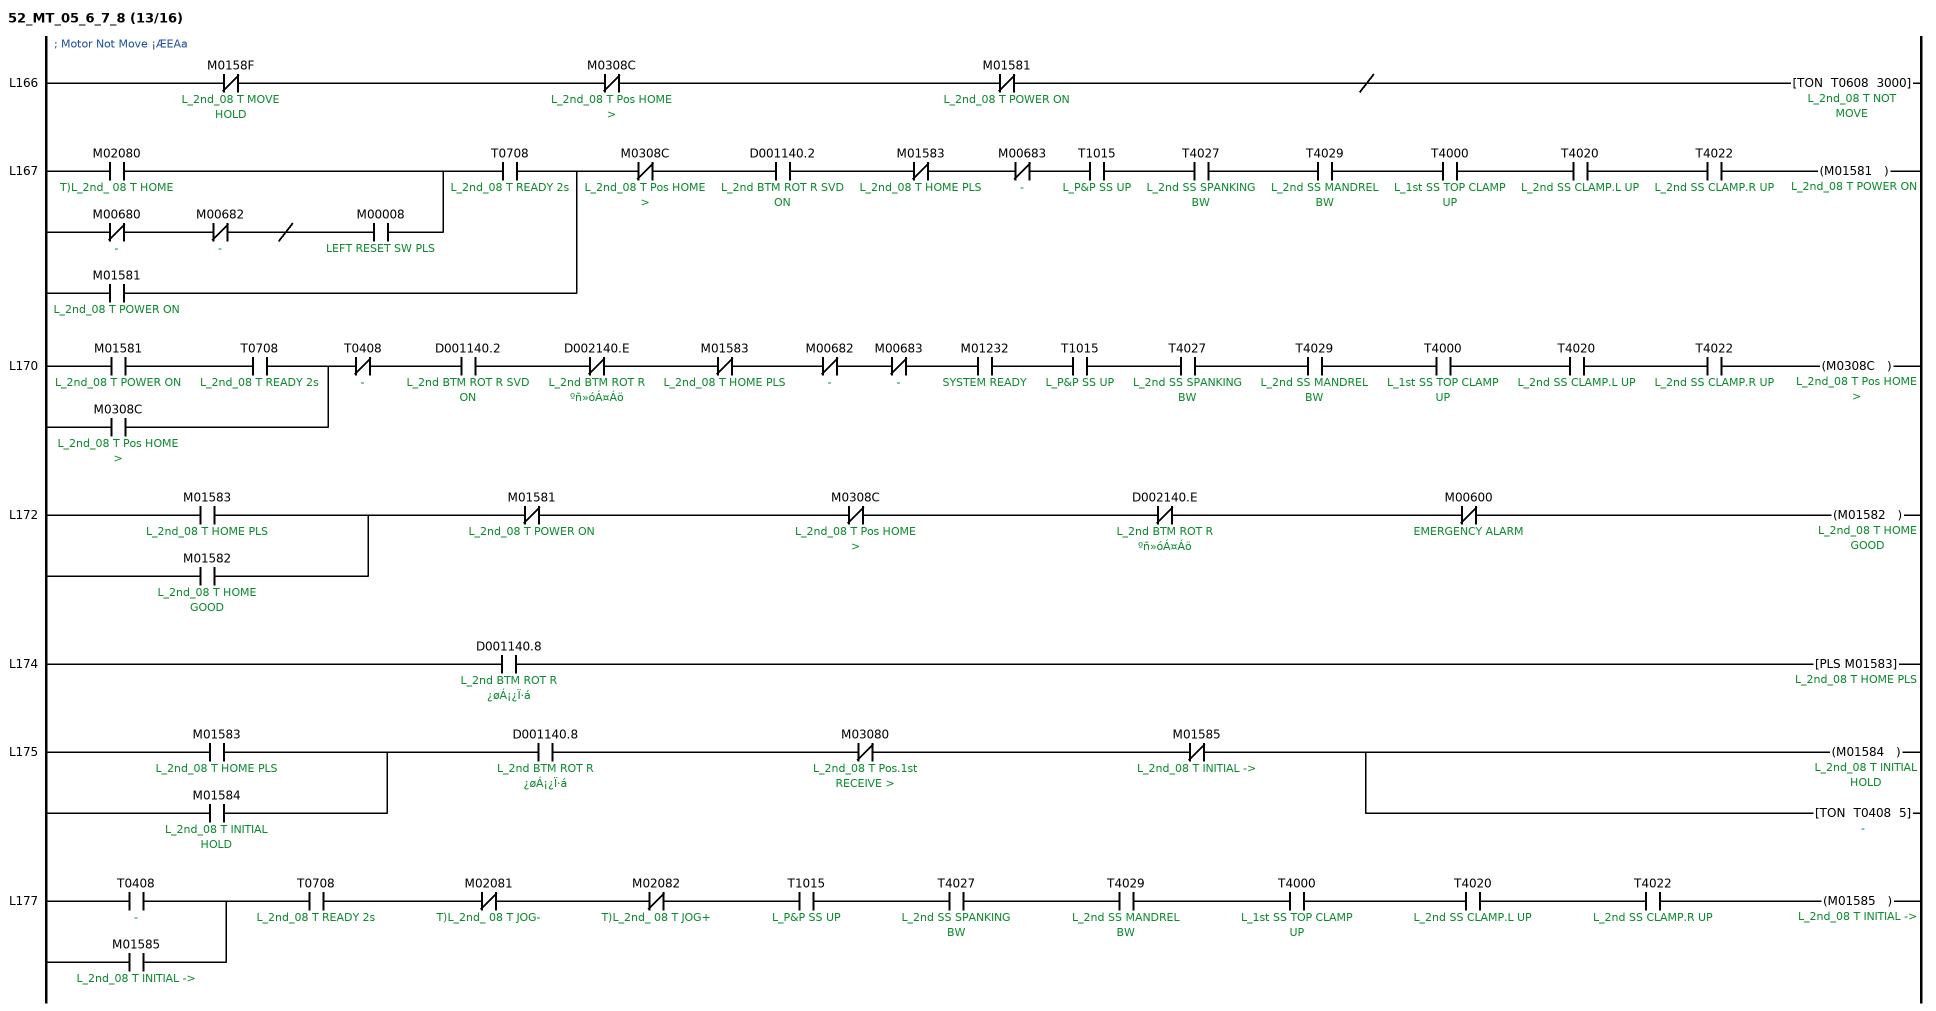
[picture p288: 52_MT_05_6_7_8 rungs L166-L177]
; L166
LOAD NOT  M0158F	// L_2nd_08 T MOVE HOLD
AND NOT   M0308C	// L_2nd_08 T Pos HOME >
AND NOT   M01581	// L_2nd_08 T POWER ON
NOT
TON       T0608 3000	// L_2nd_08 T NOT MOVE
// output comment: Motor Not Move ¡ÆEAa
; L167
LOAD      M02080	// T)L_2nd_ 08 T HOME
LOAD NOT  M00680	// -
AND NOT   M00682	// -
NOT
AND       M00008	// LEFT RESET SW PLS
OR LOAD
AND       T0708	// L_2nd_08 T READY 2s
OR        M01581	// L_2nd_08 T POWER ON
AND NOT   M0308C	// L_2nd_08 T Pos HOME >
AND       D001140.2	// L_2nd BTM ROT R SVD ON
AND NOT   M01583	// L_2nd_08 T HOME PLS
AND NOT   M00683	// -
AND       T1015	// L_P&P SS UP
AND       T4027	// L_2nd SS SPANKING BW
AND       T4029	// L_2nd SS MANDREL BW
AND       T4000	// L_1st SS TOP CLAMP    UP
AND       T4020	// L_2nd SS CLAMP.L UP
AND       T4022	// L_2nd SS CLAMP.R UP
OUT       M01581	// L_2nd_08 T POWER ON
; L170
LOAD      M01581	// L_2nd_08 T POWER ON
AND       T0708	// L_2nd_08 T READY 2s
OR        M0308C	// L_2nd_08 T Pos HOME >
AND NOT   T0408	// -
AND       D001140.2	// L_2nd BTM ROT R SVD ON
AND NOT   D002140.E	// L_2nd BTM ROT R ºñ»óÁ¤Áö
AND NOT   M01583	// L_2nd_08 T HOME PLS
AND NOT   M00682	// -
AND NOT   M00683	// -
AND       M01232	// SYSTEM READY
AND       T1015	// L_P&P SS UP
AND       T4027	// L_2nd SS SPANKING BW
AND       T4029	// L_2nd SS MANDREL BW
AND       T4000	// L_1st SS TOP CLAMP    UP
AND       T4020	// L_2nd SS CLAMP.L UP
AND       T4022	// L_2nd SS CLAMP.R UP
OUT       M0308C	// L_2nd_08 T Pos HOME >
; L172
LOAD      M01583	// L_2nd_08 T HOME PLS
OR        M01582	// L_2nd_08 T HOME GOOD
AND NOT   M01581	// L_2nd_08 T POWER ON
AND NOT   M0308C	// L_2nd_08 T Pos HOME >
AND NOT   D002140.E	// L_2nd BTM ROT R ºñ»óÁ¤Áö
AND NOT   M00600	// EMERGENCY ALARM
OUT       M01582	// L_2nd_08 T HOME GOOD
; L174
LOAD      D001140.8	// L_2nd BTM ROT R ¿øÁ¡¿Ï·á
OUTP      M01583	// L_2nd_08 T HOME PLS
; L175
LOAD      M01583	// L_2nd_08 T HOME PLS
OR        M01584	// L_2nd_08 T INITIAL HOLD
AND       D001140.8	// L_2nd BTM ROT R ¿øÁ¡¿Ï·á
AND NOT   M03080	// L_2nd_08 T Pos.1st RECEIVE >
AND NOT   M01585	// L_2nd_08 T INITIAL ->
OUT       M01584	// L_2nd_08 T INITIAL HOLD
TON       T0408 5	// -
; L177
LOAD      T0408	// -
OR        M01585	// L_2nd_08 T INITIAL ->
AND       T0708	// L_2nd_08 T READY 2s
AND NOT   M02081	// T)L_2nd_ 08 T JOG-
AND NOT   M02082	// T)L_2nd_ 08 T JOG+
AND       T1015	// L_P&P SS UP
AND       T4027	// L_2nd SS SPANKING BW
AND       T4029	// L_2nd SS MANDREL BW
AND       T4000	// L_1st SS TOP CLAMP    UP
AND       T4020	// L_2nd SS CLAMP.L UP
AND       T4022	// L_2nd SS CLAMP.R UP
OUT       M01585	// L_2nd_08 T INITIAL ->

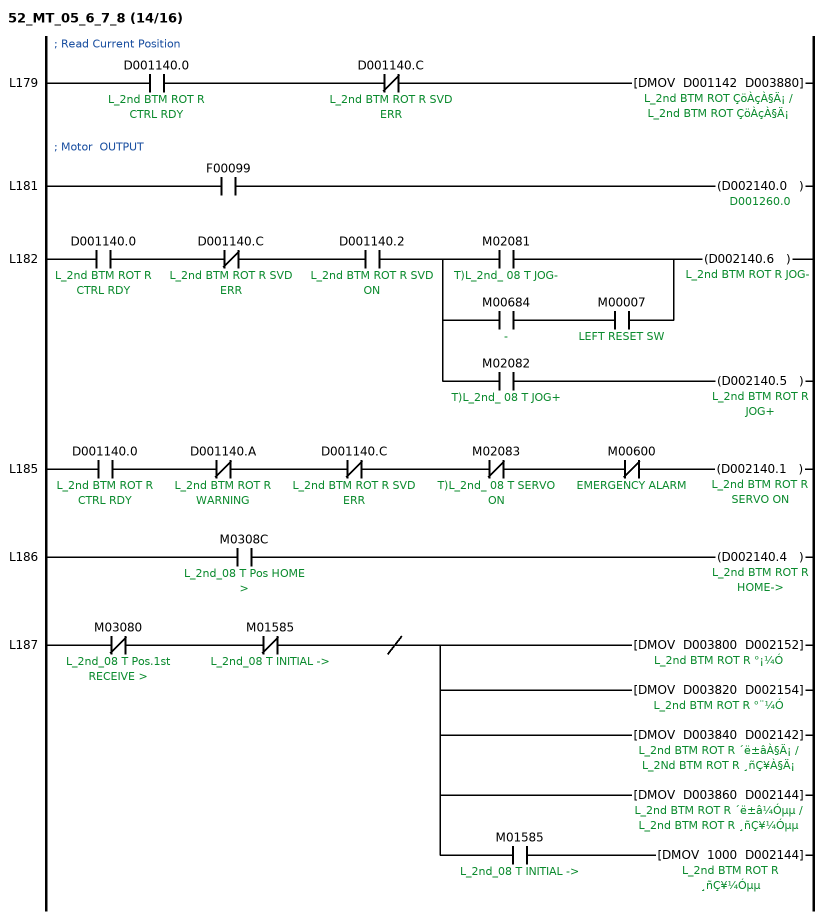
; L179
LOAD      D001140.0	// L_2nd BTM ROT R CTRL RDY
AND NOT   D001140.C	// L_2nd BTM ROT R SVD ERR
DMOV      D001142 D003880	// L_2nd BTM ROT ÇöÀçÀ§Ä¡ / L_2nd BTM ROT ÇöÀçÀ§Ä¡
// output comment: Read Current Position
//  Motor  OUTPUT
; L181
LOAD      F00099
OUT       D002140.0	// D001260.0
; L182
LOAD      D001140.0	// L_2nd BTM ROT R CTRL RDY
AND NOT   D001140.C	// L_2nd BTM ROT R SVD ERR
AND       D001140.2	// L_2nd BTM ROT R SVD ON
MPUSH
LOAD      M02081	// T)L_2nd_ 08 T JOG-
LOAD      M00684	// -
AND       M00007	// LEFT RESET SW
OR LOAD
AND LOAD
OUT       D002140.6	// L_2nd BTM ROT R JOG-
MPOP
AND       M02082	// T)L_2nd_ 08 T JOG+
OUT       D002140.5	// L_2nd BTM ROT R JOG+
; L185
LOAD      D001140.0	// L_2nd BTM ROT R CTRL RDY
AND NOT   D001140.A	// L_2nd BTM ROT R WARNING
AND NOT   D001140.C	// L_2nd BTM ROT R SVD ERR
AND NOT   M02083	// T)L_2nd_ 08 T SERVO ON
AND NOT   M00600	// EMERGENCY ALARM
OUT       D002140.1	// L_2nd BTM ROT R SERVO ON
; L186
LOAD      M0308C	// L_2nd_08 T Pos HOME >
OUT       D002140.4	// L_2nd BTM ROT R HOME->
; L187
LOAD NOT  M03080	// L_2nd_08 T Pos.1st RECEIVE >
AND NOT   M01585	// L_2nd_08 T INITIAL ->
NOT
DMOV      D003800 D002152	// L_2nd BTM ROT R °¡¼Ó
DMOV      D003820 D002154	// L_2nd BTM ROT R °¨¼Ó
DMOV      D003840 D002142	// L_2nd BTM ROT R ´ë±âÀ§Ä¡ / L_2Nd BTM ROT R ¸ñÇ¥À§Ä¡
DMOV      D003860 D002144	// L_2nd BTM ROT R ´ë±â¼Óµµ / L_2nd BTM ROT R ¸ñÇ¥¼Óµµ
AND       M01585	// L_2nd_08 T INITIAL ->
DMOV      1000 D002144	// L_2nd BTM ROT R ¸ñÇ¥¼Óµµ

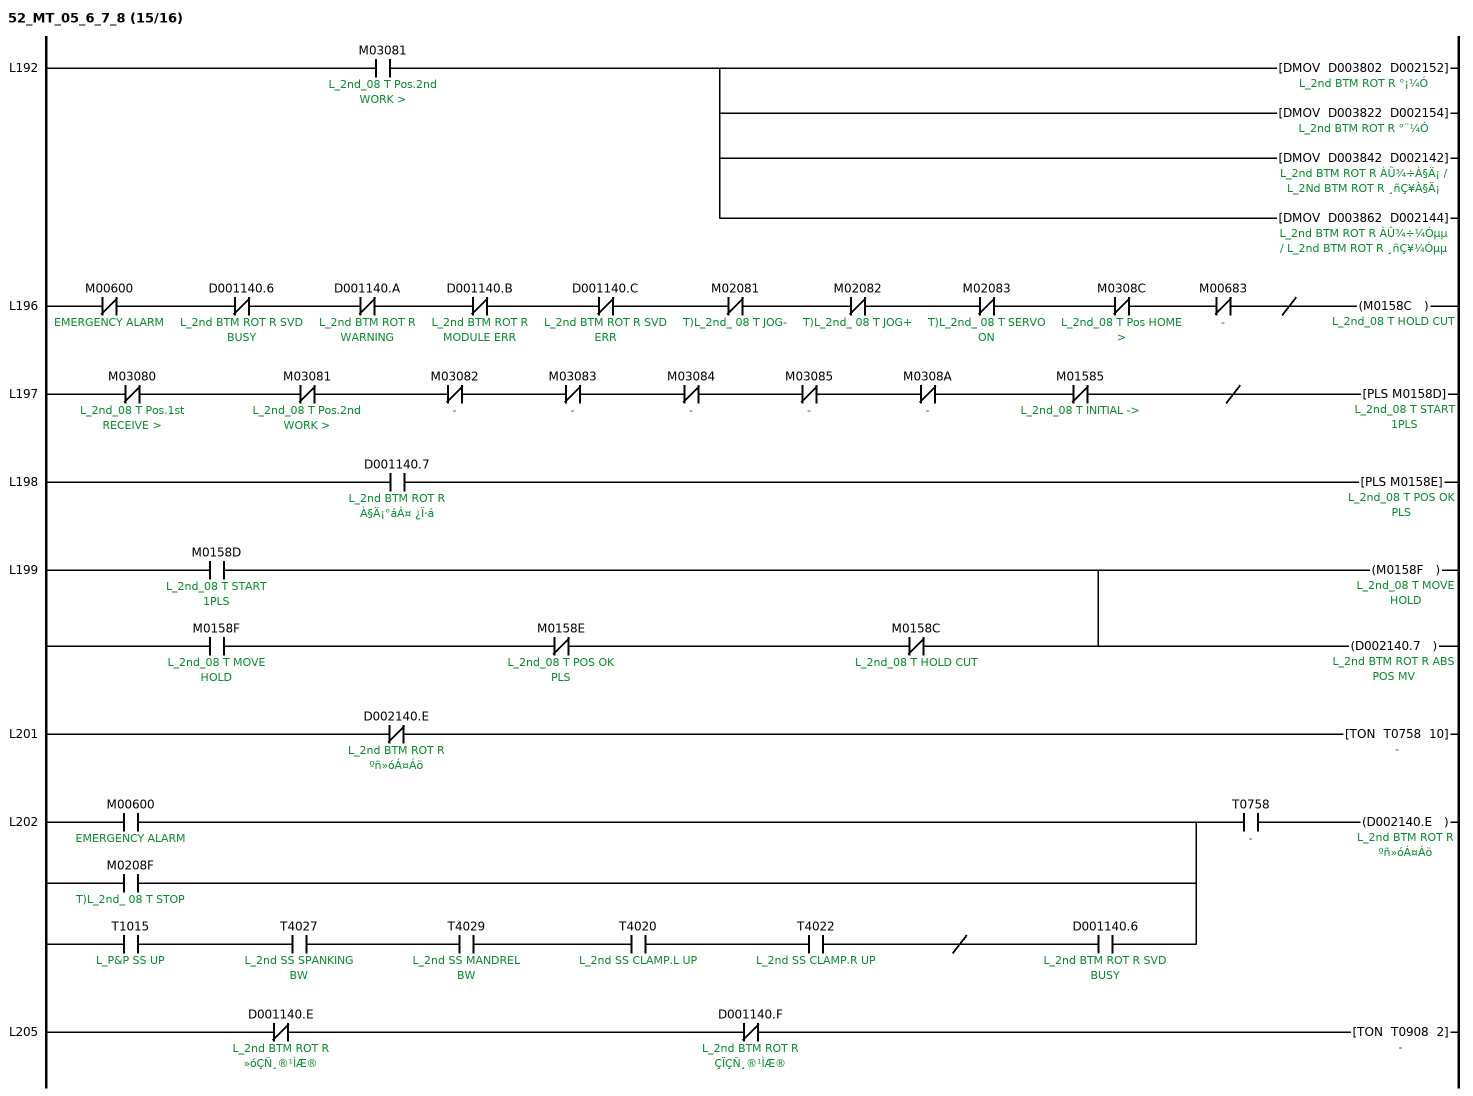
; L192
LOAD      M03081	// L_2nd_08 T Pos.2nd WORK >
DMOV      D003802 D002152	// L_2nd BTM ROT R °¡¼Ó
DMOV      D003822 D002154	// L_2nd BTM ROT R °¨¼Ó
DMOV      D003842 D002142	// L_2nd BTM ROT R ÀÛ¾÷À§Ä¡ / L_2Nd BTM ROT R ¸ñÇ¥À§Ä¡
DMOV      D003862 D002144	// L_2nd BTM ROT R ÀÛ¾÷¼Óµµ / L_2nd BTM ROT R ¸ñÇ¥¼Óµµ
; L196
LOAD NOT  M00600	// EMERGENCY ALARM
AND NOT   D001140.6	// L_2nd BTM ROT R SVD BUSY
AND NOT   D001140.A	// L_2nd BTM ROT R WARNING
AND NOT   D001140.B	// L_2nd BTM ROT R MODULE ERR
AND NOT   D001140.C	// L_2nd BTM ROT R SVD ERR
AND NOT   M02081	// T)L_2nd_ 08 T JOG-
AND NOT   M02082	// T)L_2nd_ 08 T JOG+
AND NOT   M02083	// T)L_2nd_ 08 T SERVO ON
AND NOT   M0308C	// L_2nd_08 T Pos HOME >
AND NOT   M00683	// -
NOT
OUT       M0158C	// L_2nd_08 T HOLD CUT
; L197
LOAD NOT  M03080	// L_2nd_08 T Pos.1st RECEIVE >
AND NOT   M03081	// L_2nd_08 T Pos.2nd WORK >
AND NOT   M03082	// -
AND NOT   M03083	// -
AND NOT   M03084	// -
AND NOT   M03085	// -
AND NOT   M0308A	// -
AND NOT   M01585	// L_2nd_08 T INITIAL ->
NOT
OUTP      M0158D	// L_2nd_08 T START 1PLS
; L198
LOAD      D001140.7	// L_2nd BTM ROT R À§Ä¡°áÁ¤ ¿Ï·á
OUTP      M0158E	// L_2nd_08 T POS OK PLS
; L199
LOAD      M0158D	// L_2nd_08 T START 1PLS
LOAD      M0158F	// L_2nd_08 T MOVE HOLD
AND NOT   M0158E	// L_2nd_08 T POS OK PLS
AND NOT   M0158C	// L_2nd_08 T HOLD CUT
OR LOAD
OUT       M0158F	// L_2nd_08 T MOVE HOLD
OUT       D002140.7	// L_2nd BTM ROT R ABS POS MV
; L201
LOAD NOT  D002140.E	// L_2nd BTM ROT R ºñ»óÁ¤Áö
TON       T0758 10	// -
; L202
LOAD      M00600	// EMERGENCY ALARM
OR        M0208F	// T)L_2nd_ 08 T STOP
LOAD      T1015	// L_P&P SS UP
AND       T4027	// L_2nd SS SPANKING BW
AND       T4029	// L_2nd SS MANDREL BW
AND       T4020	// L_2nd SS CLAMP.L UP
AND       T4022	// L_2nd SS CLAMP.R UP
NOT
AND       D001140.6	// L_2nd BTM ROT R SVD BUSY
OR LOAD
AND       T0758	// -
OUT       D002140.E	// L_2nd BTM ROT R ºñ»óÁ¤Áö
; L205
LOAD NOT  D001140.E	// L_2nd BTM ROT R »óÇÑ¸®¹ÌÆ®
AND NOT   D001140.F	// L_2nd BTM ROT R ÇÏÇÑ¸®¹ÌÆ®
TON       T0908 2	// -

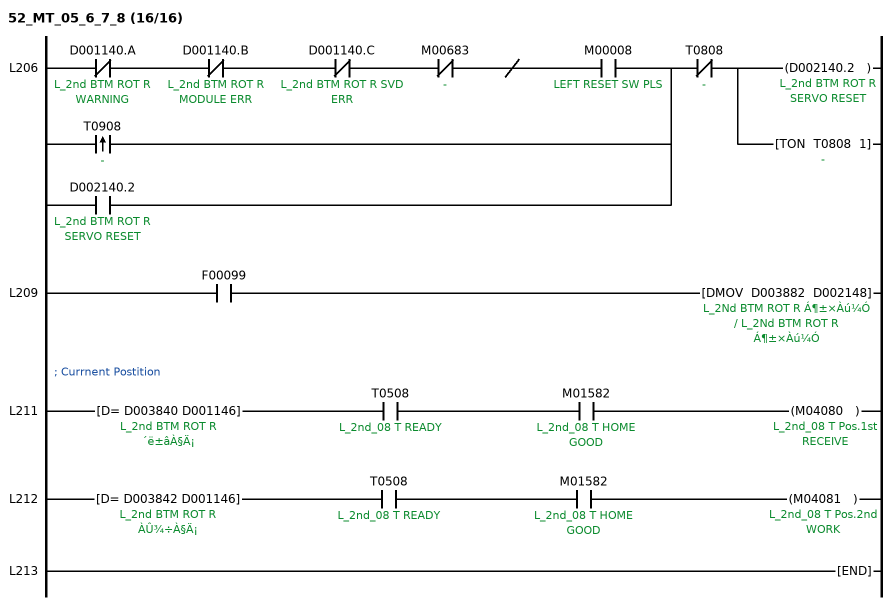
; L206
LOAD NOT  D001140.A	// L_2nd BTM ROT R WARNING
AND NOT   D001140.B	// L_2nd BTM ROT R MODULE ERR
AND NOT   D001140.C	// L_2nd BTM ROT R SVD ERR
AND NOT   M00683	// -
NOT
AND       M00008	// LEFT RESET SW PLS
ORP       T0908	// -
OR        D002140.2	// L_2nd BTM ROT R SERVO RESET
AND NOT   T0808	// -
OUT       D002140.2	// L_2nd BTM ROT R SERVO RESET
TON       T0808 1	// -
; L209
LOAD      F00099
DMOV      D003882 D002148	// L_2Nd BTM ROT R Á¶±×Àú¼Ó / L_2Nd BTM ROT R Á¶±×Àú¼Ó
// Currnent Postition
; L211
LOADD=    D003840 D001146	// L_2nd BTM ROT R ´ë±âÀ§Ä¡
AND       T0508	// L_2nd_08 T READY
AND       M01582	// L_2nd_08 T HOME GOOD
OUT       M04080	// L_2nd_08 T Pos.1st RECEIVE
; L212
LOADD=    D003842 D001146	// L_2nd BTM ROT R ÀÛ¾÷À§Ä¡
AND       T0508	// L_2nd_08 T READY
AND       M01582	// L_2nd_08 T HOME GOOD
OUT       M04081	// L_2nd_08 T Pos.2nd WORK
; L213
END

PROGRAM 53_MT_09_10_11_12 (task: ½ºÄµ ÇÁ·Î±×·¥)

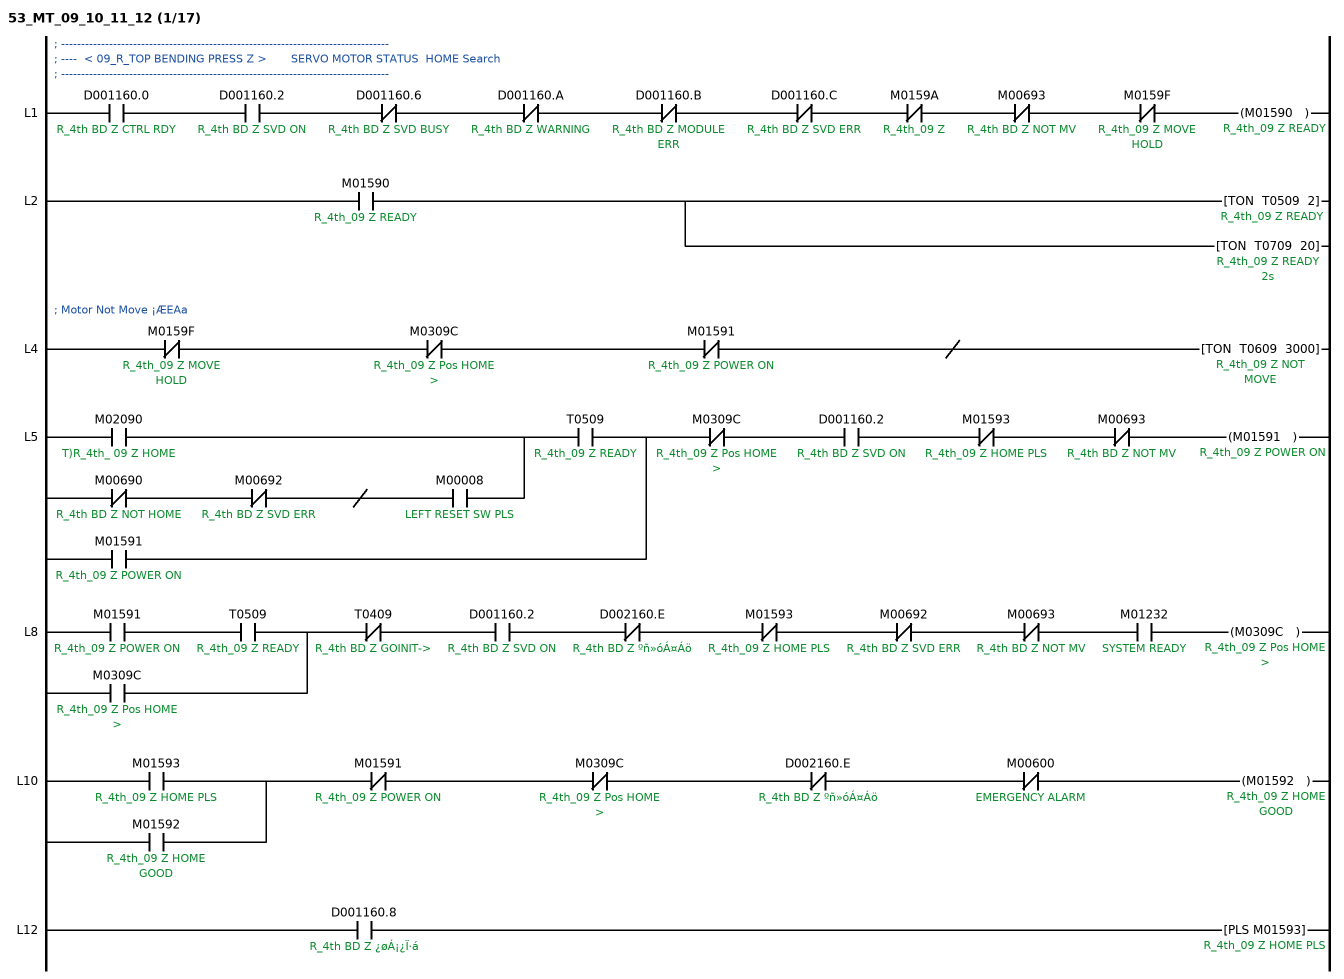
// ----------------------------------------------------------------------------------
// 
// ----  < 09_R_TOP BENDING PRESS Z >       SERVO MOTOR STATUS  HOME Search
// 
// ----------------------------------------------------------------------------------
; L1
LOAD      D001160.0	// R_4th BD Z CTRL RDY
AND       D001160.2	// R_4th BD Z SVD ON
AND NOT   D001160.6	// R_4th BD Z SVD BUSY
AND NOT   D001160.A	// R_4th BD Z WARNING
AND NOT   D001160.B	// R_4th BD Z MODULE ERR
AND NOT   D001160.C	// R_4th BD Z SVD ERR
AND NOT   M0159A	// R_4th_09 Z
AND NOT   M00693	// R_4th BD Z NOT MV
AND NOT   M0159F	// R_4th_09 Z MOVE HOLD
OUT       M01590	// R_4th_09 Z READY
; L2
LOAD      M01590	// R_4th_09 Z READY
TON       T0509 2	// R_4th_09 Z READY
TON       T0709 20	// R_4th_09 Z READY 2s
; L4
LOAD NOT  M0159F	// R_4th_09 Z MOVE HOLD
AND NOT   M0309C	// R_4th_09 Z Pos HOME >
AND NOT   M01591	// R_4th_09 Z POWER ON
NOT
TON       T0609 3000	// R_4th_09 Z NOT MOVE
// output comment: Motor Not Move ¡ÆEAa
; L5
LOAD      M02090	// T)R_4th_ 09 Z HOME
LOAD NOT  M00690	// R_4th BD Z NOT HOME
AND NOT   M00692	// R_4th BD Z SVD ERR
NOT
AND       M00008	// LEFT RESET SW PLS
OR LOAD
AND       T0509	// R_4th_09 Z READY
OR        M01591	// R_4th_09 Z POWER ON
AND NOT   M0309C	// R_4th_09 Z Pos HOME >
AND       D001160.2	// R_4th BD Z SVD ON
AND NOT   M01593	// R_4th_09 Z HOME PLS
AND NOT   M00693	// R_4th BD Z NOT MV
OUT       M01591	// R_4th_09 Z POWER ON
; L8
LOAD      M01591	// R_4th_09 Z POWER ON
AND       T0509	// R_4th_09 Z READY
OR        M0309C	// R_4th_09 Z Pos HOME >
AND NOT   T0409	// R_4th BD Z GOINIT->
AND       D001160.2	// R_4th BD Z SVD ON
AND NOT   D002160.E	// R_4th BD Z ºñ»óÁ¤Áö
AND NOT   M01593	// R_4th_09 Z HOME PLS
AND NOT   M00692	// R_4th BD Z SVD ERR
AND NOT   M00693	// R_4th BD Z NOT MV
AND       M01232	// SYSTEM READY
OUT       M0309C	// R_4th_09 Z Pos HOME >
; L10
LOAD      M01593	// R_4th_09 Z HOME PLS
OR        M01592	// R_4th_09 Z HOME GOOD
AND NOT   M01591	// R_4th_09 Z POWER ON
AND NOT   M0309C	// R_4th_09 Z Pos HOME >
AND NOT   D002160.E	// R_4th BD Z ºñ»óÁ¤Áö
AND NOT   M00600	// EMERGENCY ALARM
OUT       M01592	// R_4th_09 Z HOME GOOD
; L12
LOAD      D001160.8	// R_4th BD Z ¿øÁ¡¿Ï·á
OUTP      M01593	// R_4th_09 Z HOME PLS

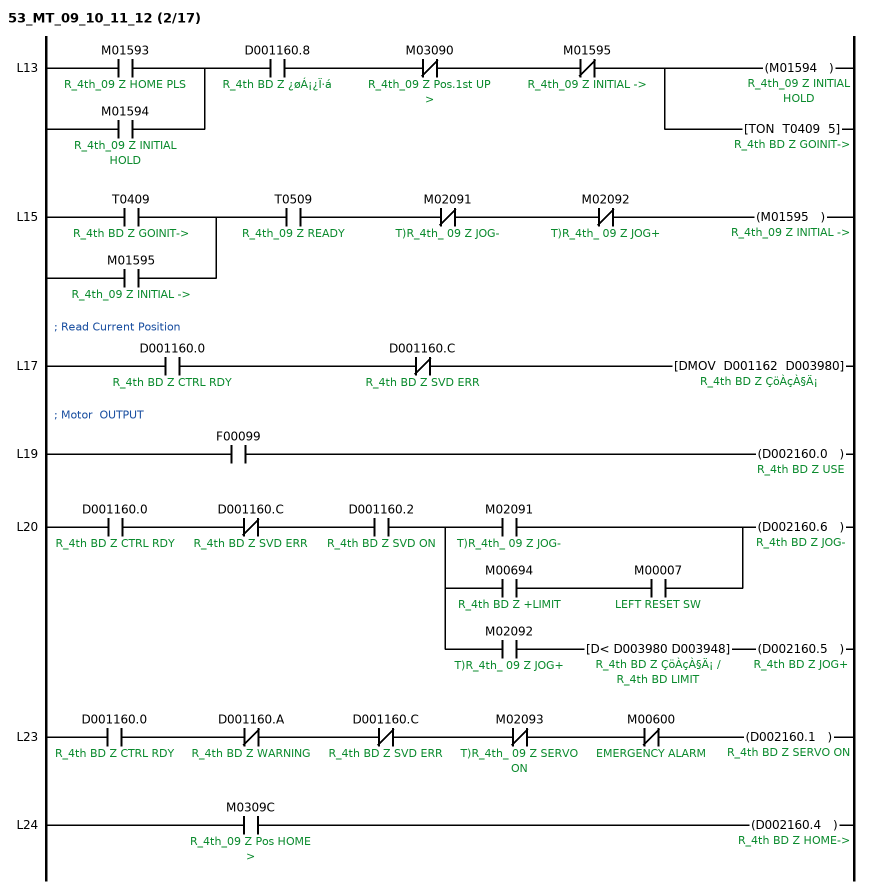
; L13
LOAD      M01593	// R_4th_09 Z HOME PLS
OR        M01594	// R_4th_09 Z INITIAL HOLD
AND       D001160.8	// R_4th BD Z ¿øÁ¡¿Ï·á
AND NOT   M03090	// R_4th_09 Z Pos.1st UP >
AND NOT   M01595	// R_4th_09 Z INITIAL ->
OUT       M01594	// R_4th_09 Z INITIAL HOLD
TON       T0409 5	// R_4th BD Z GOINIT->
; L15
LOAD      T0409	// R_4th BD Z GOINIT->
OR        M01595	// R_4th_09 Z INITIAL ->
AND       T0509	// R_4th_09 Z READY
AND NOT   M02091	// T)R_4th_ 09 Z JOG-
AND NOT   M02092	// T)R_4th_ 09 Z JOG+
OUT       M01595	// R_4th_09 Z INITIAL ->
; L17
LOAD      D001160.0	// R_4th BD Z CTRL RDY
AND NOT   D001160.C	// R_4th BD Z SVD ERR
DMOV      D001162 D003980	// R_4th BD Z ÇöÀçÀ§Ä¡
// output comment: Read Current Position
//  Motor  OUTPUT
; L19
LOAD      F00099
OUT       D002160.0	// R_4th BD Z USE
; L20
LOAD      D001160.0	// R_4th BD Z CTRL RDY
AND NOT   D001160.C	// R_4th BD Z SVD ERR
AND       D001160.2	// R_4th BD Z SVD ON
MPUSH
LOAD      M02091	// T)R_4th_ 09 Z JOG-
LOAD      M00694	// R_4th BD Z +LIMIT
AND       M00007	// LEFT RESET SW
OR LOAD
AND LOAD
OUT       D002160.6	// R_4th BD Z JOG-
MPOP
AND       M02092	// T)R_4th_ 09 Z JOG+
ANDD<     D003980 D003948	// R_4th BD Z ÇöÀçÀ§Ä¡ / R_4th BD LIMIT
OUT       D002160.5	// R_4th BD Z JOG+
; L23
LOAD      D001160.0	// R_4th BD Z CTRL RDY
AND NOT   D001160.A	// R_4th BD Z WARNING
AND NOT   D001160.C	// R_4th BD Z SVD ERR
AND NOT   M02093	// T)R_4th_ 09 Z SERVO ON
AND NOT   M00600	// EMERGENCY ALARM
OUT       D002160.1	// R_4th BD Z SERVO ON
; L24
LOAD      M0309C	// R_4th_09 Z Pos HOME >
OUT       D002160.4	// R_4th BD Z HOME->

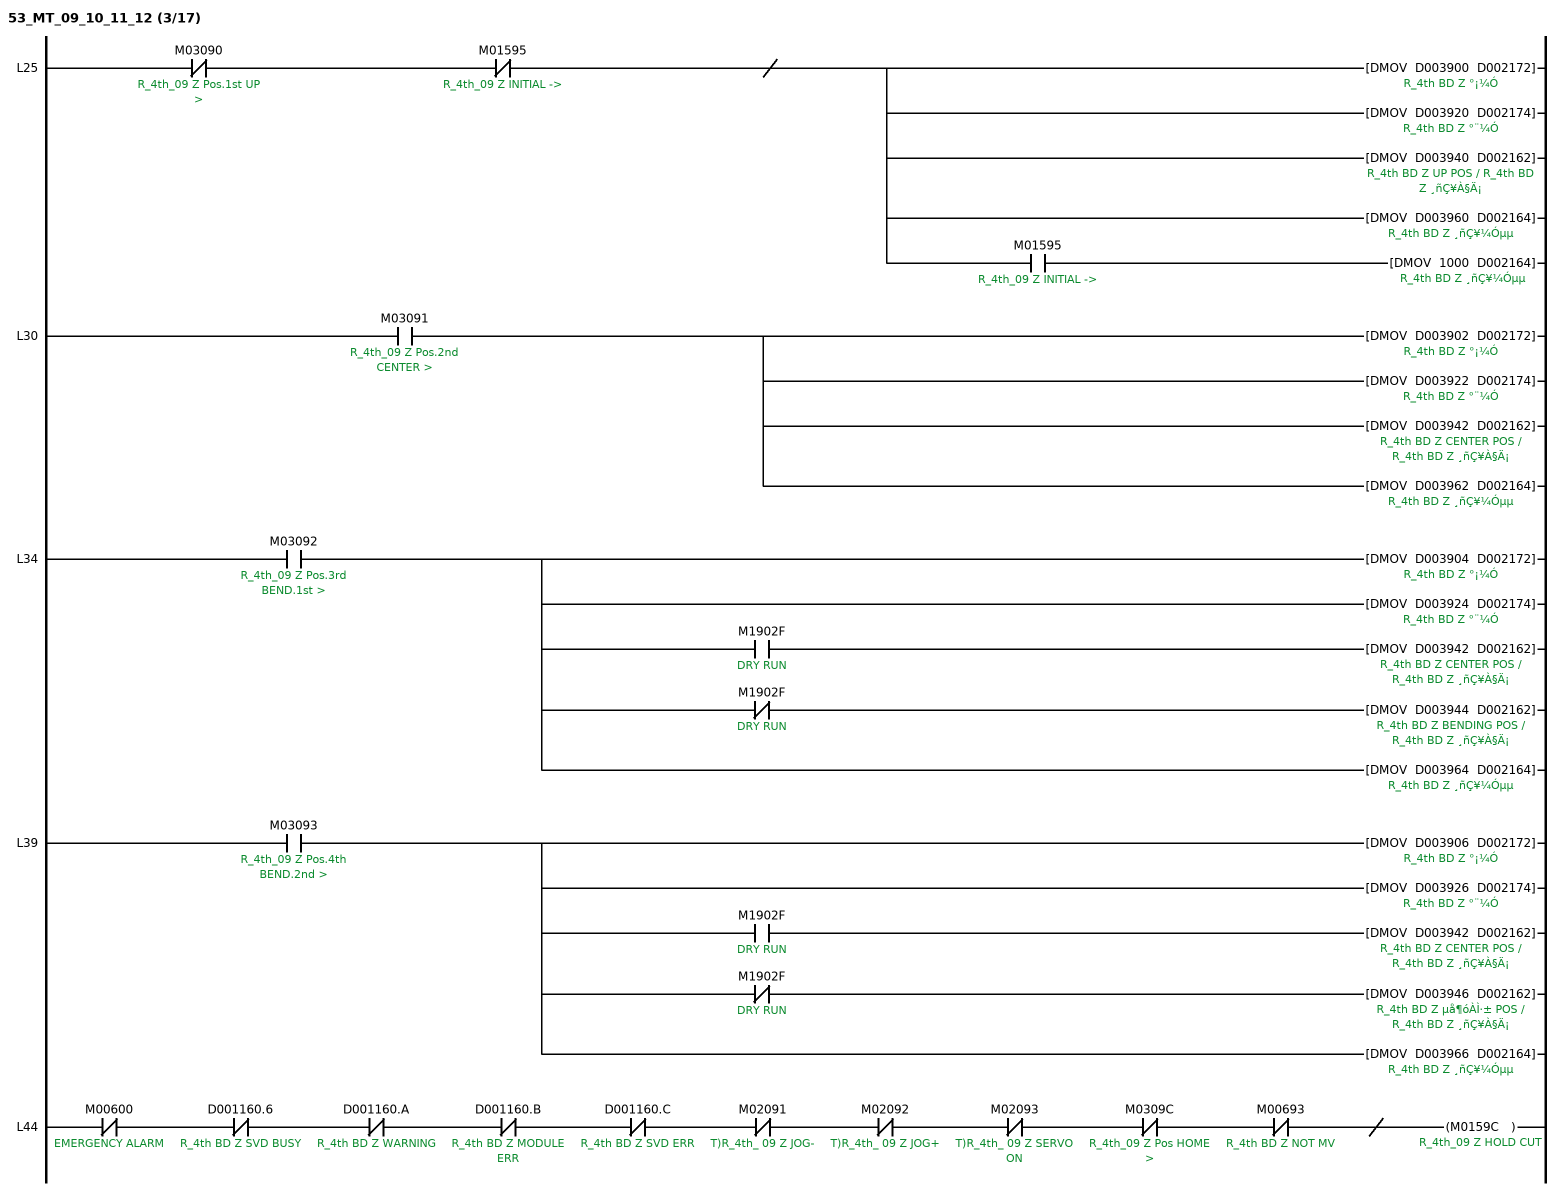
; L25
LOAD NOT  M03090	// R_4th_09 Z Pos.1st UP >
AND NOT   M01595	// R_4th_09 Z INITIAL ->
NOT
DMOV      D003900 D002172	// R_4th BD Z °¡¼Ó
DMOV      D003920 D002174	// R_4th BD Z °¨¼Ó
DMOV      D003940 D002162	// R_4th BD Z UP POS / R_4th BD Z ¸ñÇ¥À§Ä¡
DMOV      D003960 D002164	// R_4th BD Z ¸ñÇ¥¼Óµµ
AND       M01595	// R_4th_09 Z INITIAL ->
DMOV      1000 D002164	// R_4th BD Z ¸ñÇ¥¼Óµµ
; L30
LOAD      M03091	// R_4th_09 Z Pos.2nd CENTER >
DMOV      D003902 D002172	// R_4th BD Z °¡¼Ó
DMOV      D003922 D002174	// R_4th BD Z °¨¼Ó
DMOV      D003942 D002162	// R_4th BD Z CENTER POS / R_4th BD Z ¸ñÇ¥À§Ä¡
DMOV      D003962 D002164	// R_4th BD Z ¸ñÇ¥¼Óµµ
; L34
LOAD      M03092	// R_4th_09 Z Pos.3rd BEND.1st >
DMOV      D003904 D002172	// R_4th BD Z °¡¼Ó
DMOV      D003924 D002174	// R_4th BD Z °¨¼Ó
MPUSH
AND       M1902F	// DRY RUN
DMOV      D003942 D002162	// R_4th BD Z CENTER POS / R_4th BD Z ¸ñÇ¥À§Ä¡
MLOAD
AND NOT   M1902F	// DRY RUN
DMOV      D003944 D002162	// R_4th BD Z BENDING POS / R_4th BD Z ¸ñÇ¥À§Ä¡
MPOP
DMOV      D003964 D002164	// R_4th BD Z ¸ñÇ¥¼Óµµ
; L39
LOAD      M03093	// R_4th_09 Z Pos.4th BEND.2nd >
DMOV      D003906 D002172	// R_4th BD Z °¡¼Ó
DMOV      D003926 D002174	// R_4th BD Z °¨¼Ó
MPUSH
AND       M1902F	// DRY RUN
DMOV      D003942 D002162	// R_4th BD Z CENTER POS / R_4th BD Z ¸ñÇ¥À§Ä¡
MLOAD
AND NOT   M1902F	// DRY RUN
DMOV      D003946 D002162	// R_4th BD Z µå¶óÀÌ·± POS / R_4th BD Z ¸ñÇ¥À§Ä¡
MPOP
DMOV      D003966 D002164	// R_4th BD Z ¸ñÇ¥¼Óµµ
; L44
LOAD NOT  M00600	// EMERGENCY ALARM
AND NOT   D001160.6	// R_4th BD Z SVD BUSY
AND NOT   D001160.A	// R_4th BD Z WARNING
AND NOT   D001160.B	// R_4th BD Z MODULE ERR
AND NOT   D001160.C	// R_4th BD Z SVD ERR
AND NOT   M02091	// T)R_4th_ 09 Z JOG-
AND NOT   M02092	// T)R_4th_ 09 Z JOG+
AND NOT   M02093	// T)R_4th_ 09 Z SERVO ON
AND NOT   M0309C	// R_4th_09 Z Pos HOME >
AND NOT   M00693	// R_4th BD Z NOT MV
NOT
OUT       M0159C	// R_4th_09 Z HOLD CUT

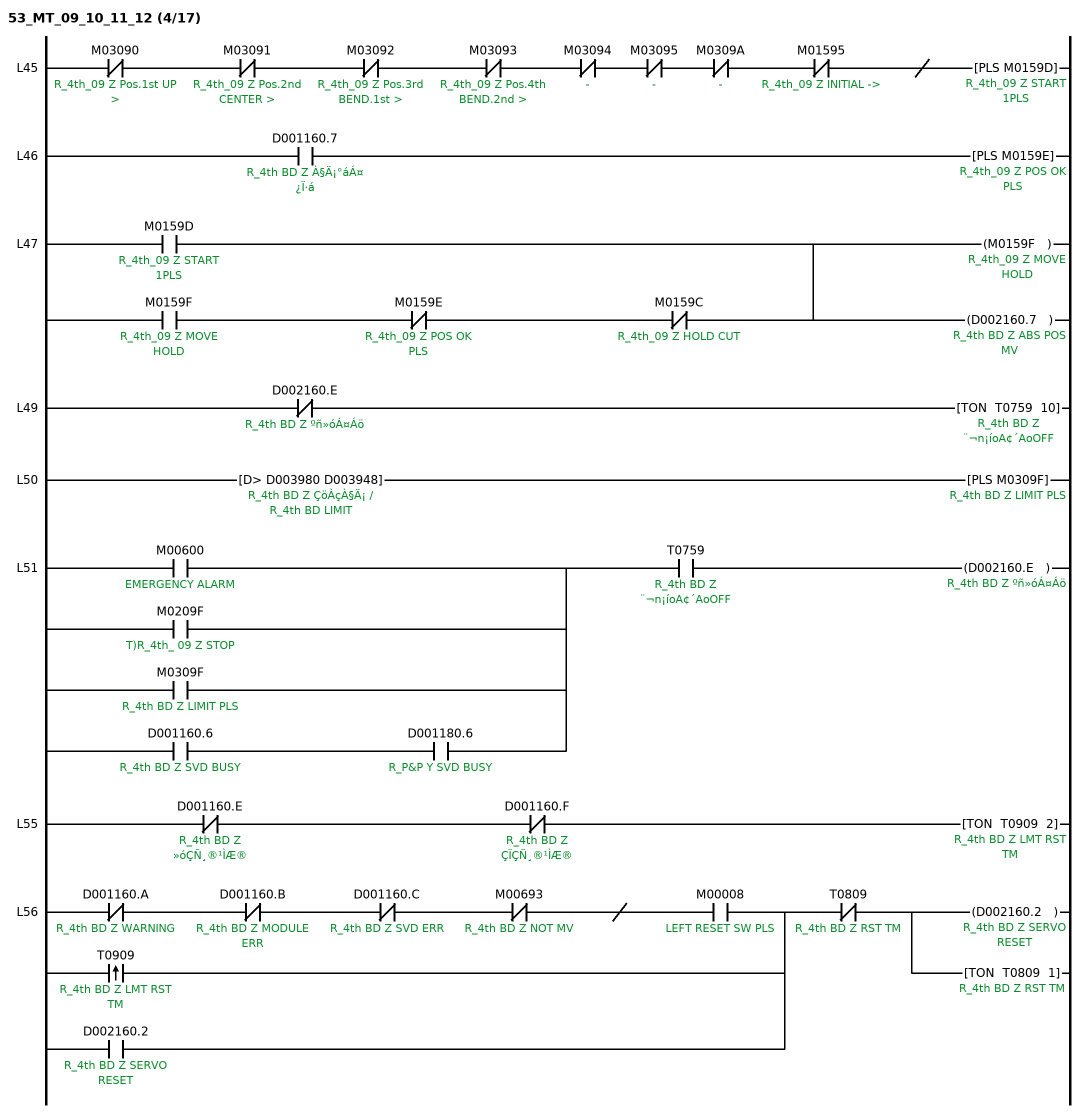
; L45
LOAD NOT  M03090	// R_4th_09 Z Pos.1st UP >
AND NOT   M03091	// R_4th_09 Z Pos.2nd CENTER >
AND NOT   M03092	// R_4th_09 Z Pos.3rd BEND.1st >
AND NOT   M03093	// R_4th_09 Z Pos.4th BEND.2nd >
AND NOT   M03094	// -
AND NOT   M03095	// -
AND NOT   M0309A	// -
AND NOT   M01595	// R_4th_09 Z INITIAL ->
NOT
OUTP      M0159D	// R_4th_09 Z START 1PLS
; L46
LOAD      D001160.7	// R_4th BD Z À§Ä¡°áÁ¤ ¿Ï·á
OUTP      M0159E	// R_4th_09 Z POS OK PLS
; L47
LOAD      M0159D	// R_4th_09 Z START 1PLS
LOAD      M0159F	// R_4th_09 Z MOVE HOLD
AND NOT   M0159E	// R_4th_09 Z POS OK PLS
AND NOT   M0159C	// R_4th_09 Z HOLD CUT
OR LOAD
OUT       M0159F	// R_4th_09 Z MOVE HOLD
OUT       D002160.7	// R_4th BD Z ABS POS MV
; L49
LOAD NOT  D002160.E	// R_4th BD Z ºñ»óÁ¤Áö
TON       T0759 10	// R_4th BD Z ¨¬n¡íoA¢´AoOFF
; L50
LOADD>    D003980 D003948	// R_4th BD Z ÇöÀçÀ§Ä¡ / R_4th BD LIMIT
OUTP      M0309F	// R_4th BD Z LIMIT PLS
; L51
LOAD      M00600	// EMERGENCY ALARM
OR        M0209F	// T)R_4th_ 09 Z STOP
OR        M0309F	// R_4th BD Z LIMIT PLS
LOAD      D001160.6	// R_4th BD Z SVD BUSY
AND       D001180.6	// R_P&P Y SVD BUSY
OR LOAD
AND       T0759	// R_4th BD Z ¨¬n¡íoA¢´AoOFF
OUT       D002160.E	// R_4th BD Z ºñ»óÁ¤Áö
; L55
LOAD NOT  D001160.E	// R_4th BD Z »óÇÑ¸®¹ÌÆ®
AND NOT   D001160.F	// R_4th BD Z ÇÏÇÑ¸®¹ÌÆ®
TON       T0909 2	// R_4th BD Z LMT RST TM
; L56
LOAD NOT  D001160.A	// R_4th BD Z WARNING
AND NOT   D001160.B	// R_4th BD Z MODULE ERR
AND NOT   D001160.C	// R_4th BD Z SVD ERR
AND NOT   M00693	// R_4th BD Z NOT MV
NOT
AND       M00008	// LEFT RESET SW PLS
ORP       T0909	// R_4th BD Z LMT RST TM
OR        D002160.2	// R_4th BD Z SERVO RESET
AND NOT   T0809	// R_4th BD Z RST TM
OUT       D002160.2	// R_4th BD Z SERVO RESET
TON       T0809 1	// R_4th BD Z RST TM

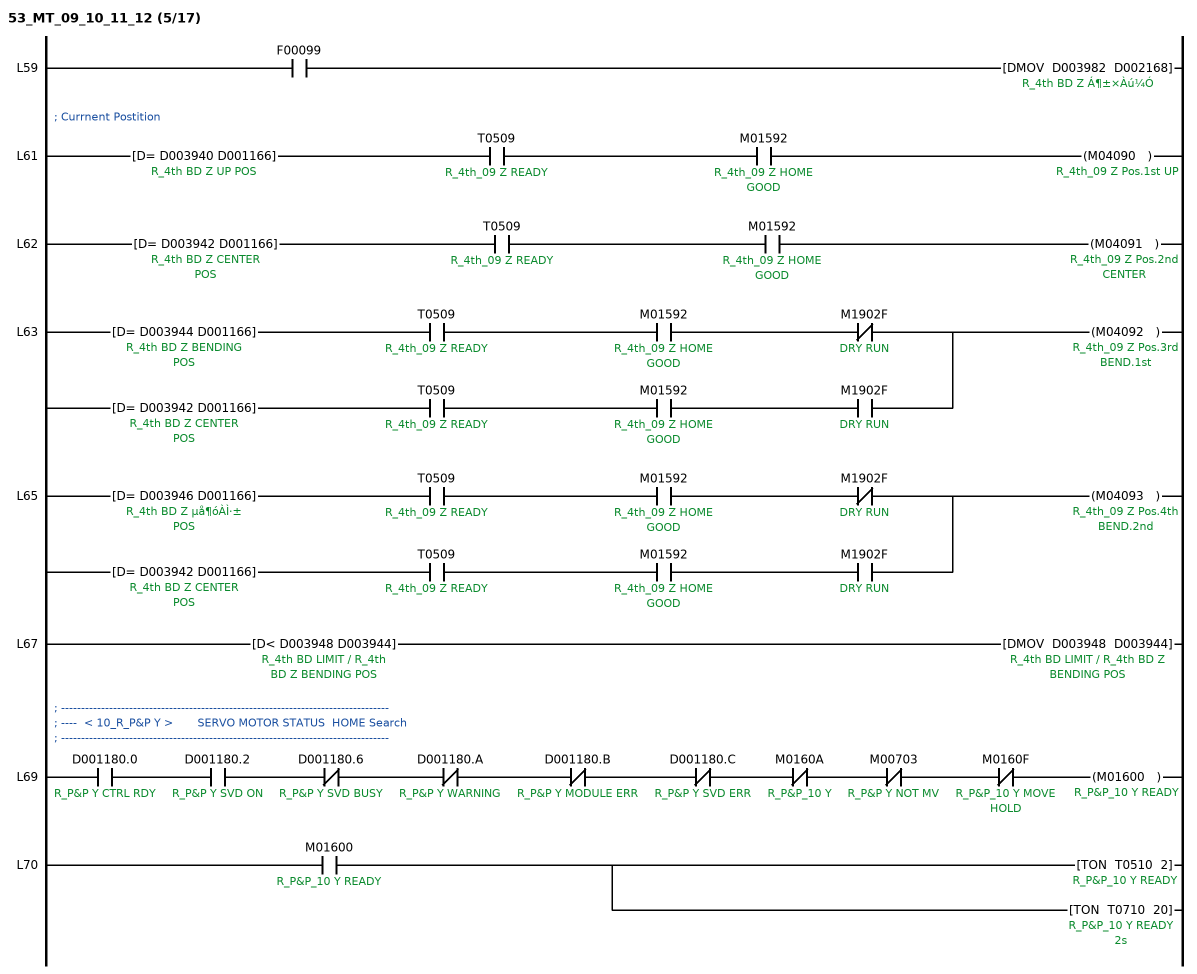
; L59
LOAD      F00099
DMOV      D003982 D002168	// R_4th BD Z Á¶±×Àú¼Ó
// Currnent Postition
; L61
LOADD=    D003940 D001166	// R_4th BD Z UP POS
AND       T0509	// R_4th_09 Z READY
AND       M01592	// R_4th_09 Z HOME GOOD
OUT       M04090	// R_4th_09 Z Pos.1st UP
; L62
LOADD=    D003942 D001166	// R_4th BD Z CENTER POS
AND       T0509	// R_4th_09 Z READY
AND       M01592	// R_4th_09 Z HOME GOOD
OUT       M04091	// R_4th_09 Z Pos.2nd CENTER
; L63
LOADD=    D003944 D001166	// R_4th BD Z BENDING POS
AND       T0509	// R_4th_09 Z READY
AND       M01592	// R_4th_09 Z HOME GOOD
AND NOT   M1902F	// DRY RUN
LOADD=    D003942 D001166	// R_4th BD Z CENTER POS
AND       T0509	// R_4th_09 Z READY
AND       M01592	// R_4th_09 Z HOME GOOD
AND       M1902F	// DRY RUN
OR LOAD
OUT       M04092	// R_4th_09 Z Pos.3rd BEND.1st
; L65
LOADD=    D003946 D001166	// R_4th BD Z µå¶óÀÌ·± POS
AND       T0509	// R_4th_09 Z READY
AND       M01592	// R_4th_09 Z HOME GOOD
AND NOT   M1902F	// DRY RUN
LOADD=    D003942 D001166	// R_4th BD Z CENTER POS
AND       T0509	// R_4th_09 Z READY
AND       M01592	// R_4th_09 Z HOME GOOD
AND       M1902F	// DRY RUN
OR LOAD
OUT       M04093	// R_4th_09 Z Pos.4th BEND.2nd
; L67
LOADD<    D003948 D003944	// R_4th BD LIMIT / R_4th BD Z BENDING POS
DMOV      D003948 D003944	// R_4th BD LIMIT / R_4th BD Z BENDING POS
// ----------------------------------------------------------------------------------
// 
// ----  < 10_R_P&P Y >       SERVO MOTOR STATUS  HOME Search
// 
// ----------------------------------------------------------------------------------
; L69
LOAD      D001180.0	// R_P&P Y CTRL RDY
AND       D001180.2	// R_P&P Y SVD ON
AND NOT   D001180.6	// R_P&P Y SVD BUSY
AND NOT   D001180.A	// R_P&P Y WARNING
AND NOT   D001180.B	// R_P&P Y MODULE ERR
AND NOT   D001180.C	// R_P&P Y SVD ERR
AND NOT   M0160A	// R_P&P_10 Y
AND NOT   M00703	// R_P&P Y NOT MV
AND NOT   M0160F	// R_P&P_10 Y MOVE HOLD
OUT       M01600	// R_P&P_10 Y READY
; L70
LOAD      M01600	// R_P&P_10 Y READY
TON       T0510 2	// R_P&P_10 Y READY
TON       T0710 20	// R_P&P_10 Y READY 2s

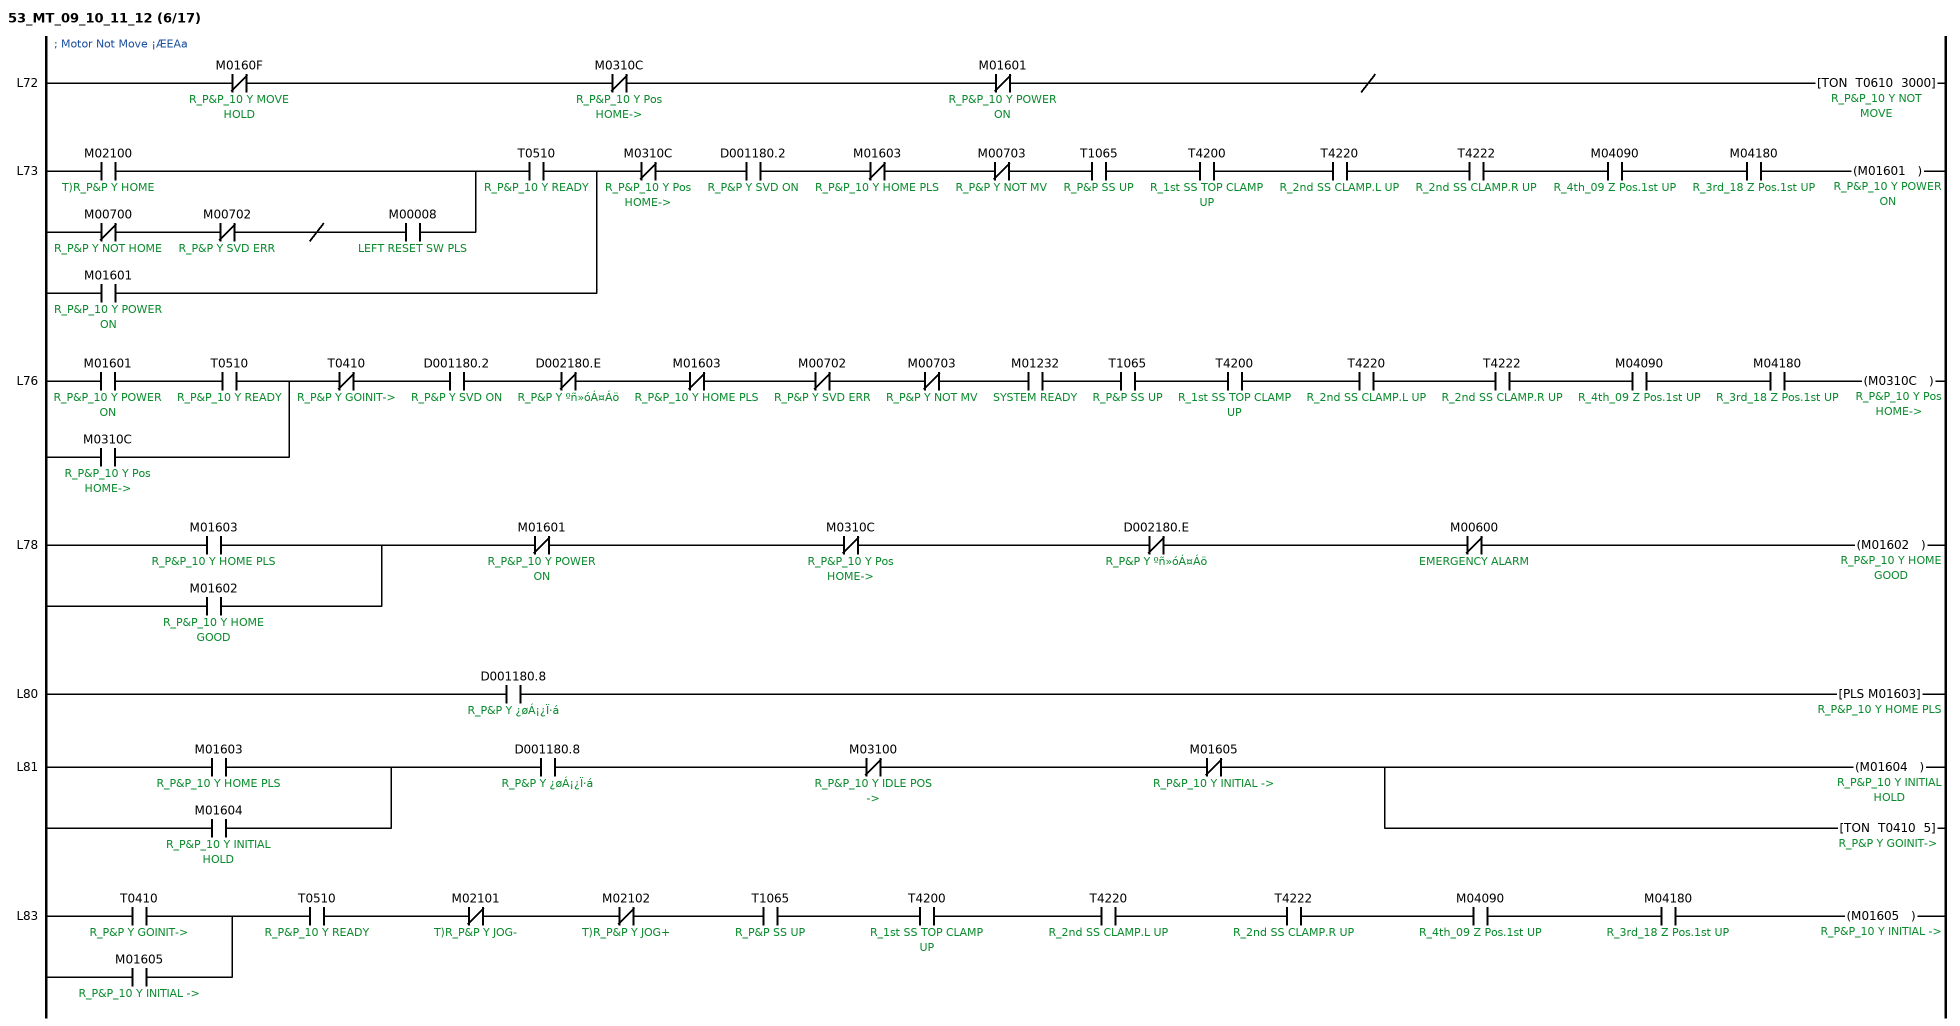
; L72
LOAD NOT  M0160F	// R_P&P_10 Y MOVE HOLD
AND NOT   M0310C	// R_P&P_10 Y Pos HOME->
AND NOT   M01601	// R_P&P_10 Y POWER ON
NOT
TON       T0610 3000	// R_P&P_10 Y NOT MOVE
// output comment: Motor Not Move ¡ÆEAa
; L73
LOAD      M02100	// T)R_P&P Y HOME
LOAD NOT  M00700	// R_P&P Y NOT HOME
AND NOT   M00702	// R_P&P Y SVD ERR
NOT
AND       M00008	// LEFT RESET SW PLS
OR LOAD
AND       T0510	// R_P&P_10 Y READY
OR        M01601	// R_P&P_10 Y POWER ON
AND NOT   M0310C	// R_P&P_10 Y Pos HOME->
AND       D001180.2	// R_P&P Y SVD ON
AND NOT   M01603	// R_P&P_10 Y HOME PLS
AND NOT   M00703	// R_P&P Y NOT MV
AND       T1065	// R_P&P SS UP
AND       T4200	// R_1st SS TOP CLAMP UP
AND       T4220	// R_2nd SS CLAMP.L UP
AND       T4222	// R_2nd SS CLAMP.R UP
AND       M04090	// R_4th_09 Z Pos.1st UP
AND       M04180	// R_3rd_18 Z Pos.1st UP
OUT       M01601	// R_P&P_10 Y POWER ON
; L76
LOAD      M01601	// R_P&P_10 Y POWER ON
AND       T0510	// R_P&P_10 Y READY
OR        M0310C	// R_P&P_10 Y Pos HOME->
AND NOT   T0410	// R_P&P Y GOINIT->
AND       D001180.2	// R_P&P Y SVD ON
AND NOT   D002180.E	// R_P&P Y ºñ»óÁ¤Áö
AND NOT   M01603	// R_P&P_10 Y HOME PLS
AND NOT   M00702	// R_P&P Y SVD ERR
AND NOT   M00703	// R_P&P Y NOT MV
AND       M01232	// SYSTEM READY
AND       T1065	// R_P&P SS UP
AND       T4200	// R_1st SS TOP CLAMP UP
AND       T4220	// R_2nd SS CLAMP.L UP
AND       T4222	// R_2nd SS CLAMP.R UP
AND       M04090	// R_4th_09 Z Pos.1st UP
AND       M04180	// R_3rd_18 Z Pos.1st UP
OUT       M0310C	// R_P&P_10 Y Pos HOME->
; L78
LOAD      M01603	// R_P&P_10 Y HOME PLS
OR        M01602	// R_P&P_10 Y HOME GOOD
AND NOT   M01601	// R_P&P_10 Y POWER ON
AND NOT   M0310C	// R_P&P_10 Y Pos HOME->
AND NOT   D002180.E	// R_P&P Y ºñ»óÁ¤Áö
AND NOT   M00600	// EMERGENCY ALARM
OUT       M01602	// R_P&P_10 Y HOME GOOD
; L80
LOAD      D001180.8	// R_P&P Y ¿øÁ¡¿Ï·á
OUTP      M01603	// R_P&P_10 Y HOME PLS
; L81
LOAD      M01603	// R_P&P_10 Y HOME PLS
OR        M01604	// R_P&P_10 Y INITIAL HOLD
AND       D001180.8	// R_P&P Y ¿øÁ¡¿Ï·á
AND NOT   M03100	// R_P&P_10 Y IDLE POS ->
AND NOT   M01605	// R_P&P_10 Y INITIAL ->
OUT       M01604	// R_P&P_10 Y INITIAL HOLD
TON       T0410 5	// R_P&P Y GOINIT->
; L83
LOAD      T0410	// R_P&P Y GOINIT->
OR        M01605	// R_P&P_10 Y INITIAL ->
AND       T0510	// R_P&P_10 Y READY
AND NOT   M02101	// T)R_P&P Y JOG-
AND NOT   M02102	// T)R_P&P Y JOG+
AND       T1065	// R_P&P SS UP
AND       T4200	// R_1st SS TOP CLAMP UP
AND       T4220	// R_2nd SS CLAMP.L UP
AND       T4222	// R_2nd SS CLAMP.R UP
AND       M04090	// R_4th_09 Z Pos.1st UP
AND       M04180	// R_3rd_18 Z Pos.1st UP
OUT       M01605	// R_P&P_10 Y INITIAL ->

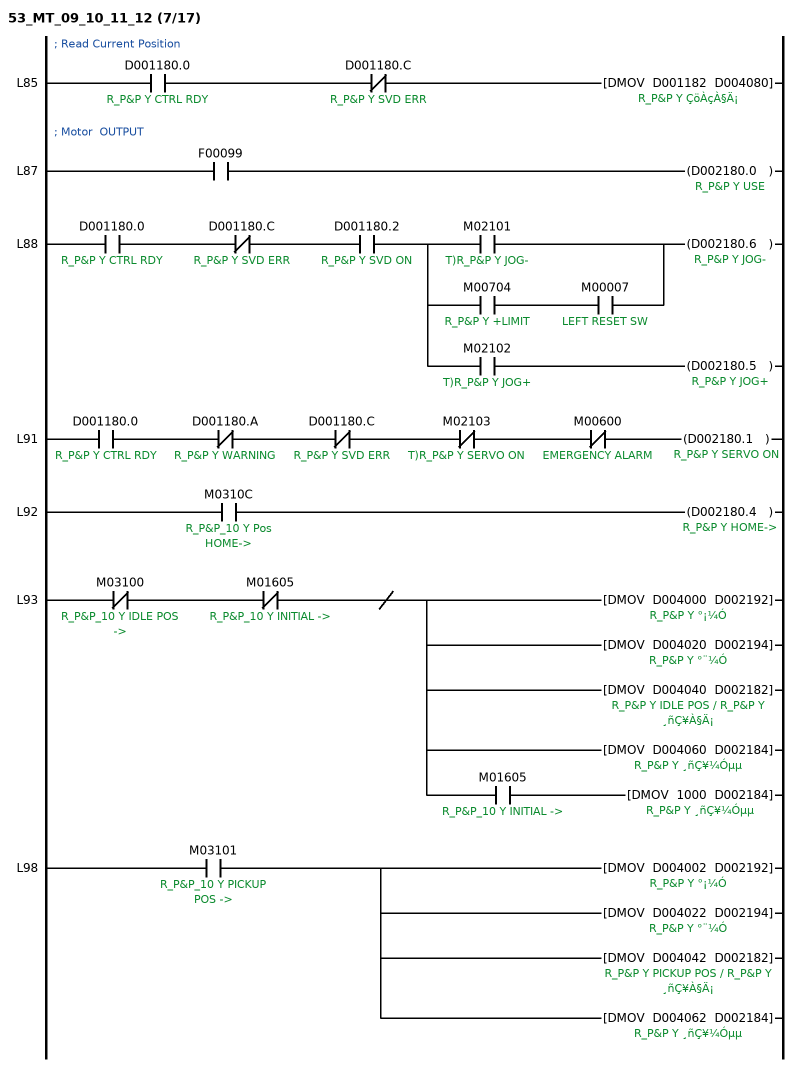
; L85
LOAD      D001180.0	// R_P&P Y CTRL RDY
AND NOT   D001180.C	// R_P&P Y SVD ERR
DMOV      D001182 D004080	// R_P&P Y ÇöÀçÀ§Ä¡
// output comment: Read Current Position
//  Motor  OUTPUT
; L87
LOAD      F00099
OUT       D002180.0	// R_P&P Y USE
; L88
LOAD      D001180.0	// R_P&P Y CTRL RDY
AND NOT   D001180.C	// R_P&P Y SVD ERR
AND       D001180.2	// R_P&P Y SVD ON
MPUSH
LOAD      M02101	// T)R_P&P Y JOG-
LOAD      M00704	// R_P&P Y +LIMIT
AND       M00007	// LEFT RESET SW
OR LOAD
AND LOAD
OUT       D002180.6	// R_P&P Y JOG-
MPOP
AND       M02102	// T)R_P&P Y JOG+
OUT       D002180.5	// R_P&P Y JOG+
; L91
LOAD      D001180.0	// R_P&P Y CTRL RDY
AND NOT   D001180.A	// R_P&P Y WARNING
AND NOT   D001180.C	// R_P&P Y SVD ERR
AND NOT   M02103	// T)R_P&P Y SERVO ON
AND NOT   M00600	// EMERGENCY ALARM
OUT       D002180.1	// R_P&P Y SERVO ON
; L92
LOAD      M0310C	// R_P&P_10 Y Pos HOME->
OUT       D002180.4	// R_P&P Y HOME->
; L93
LOAD NOT  M03100	// R_P&P_10 Y IDLE POS ->
AND NOT   M01605	// R_P&P_10 Y INITIAL ->
NOT
DMOV      D004000 D002192	// R_P&P Y °¡¼Ó
DMOV      D004020 D002194	// R_P&P Y °¨¼Ó
DMOV      D004040 D002182	// R_P&P Y IDLE POS / R_P&P Y ¸ñÇ¥À§Ä¡
DMOV      D004060 D002184	// R_P&P Y ¸ñÇ¥¼Óµµ
AND       M01605	// R_P&P_10 Y INITIAL ->
DMOV      1000 D002184	// R_P&P Y ¸ñÇ¥¼Óµµ
; L98
LOAD      M03101	// R_P&P_10 Y PICKUP POS ->
DMOV      D004002 D002192	// R_P&P Y °¡¼Ó
DMOV      D004022 D002194	// R_P&P Y °¨¼Ó
DMOV      D004042 D002182	// R_P&P Y PICKUP POS / R_P&P Y ¸ñÇ¥À§Ä¡
DMOV      D004062 D002184	// R_P&P Y ¸ñÇ¥¼Óµµ

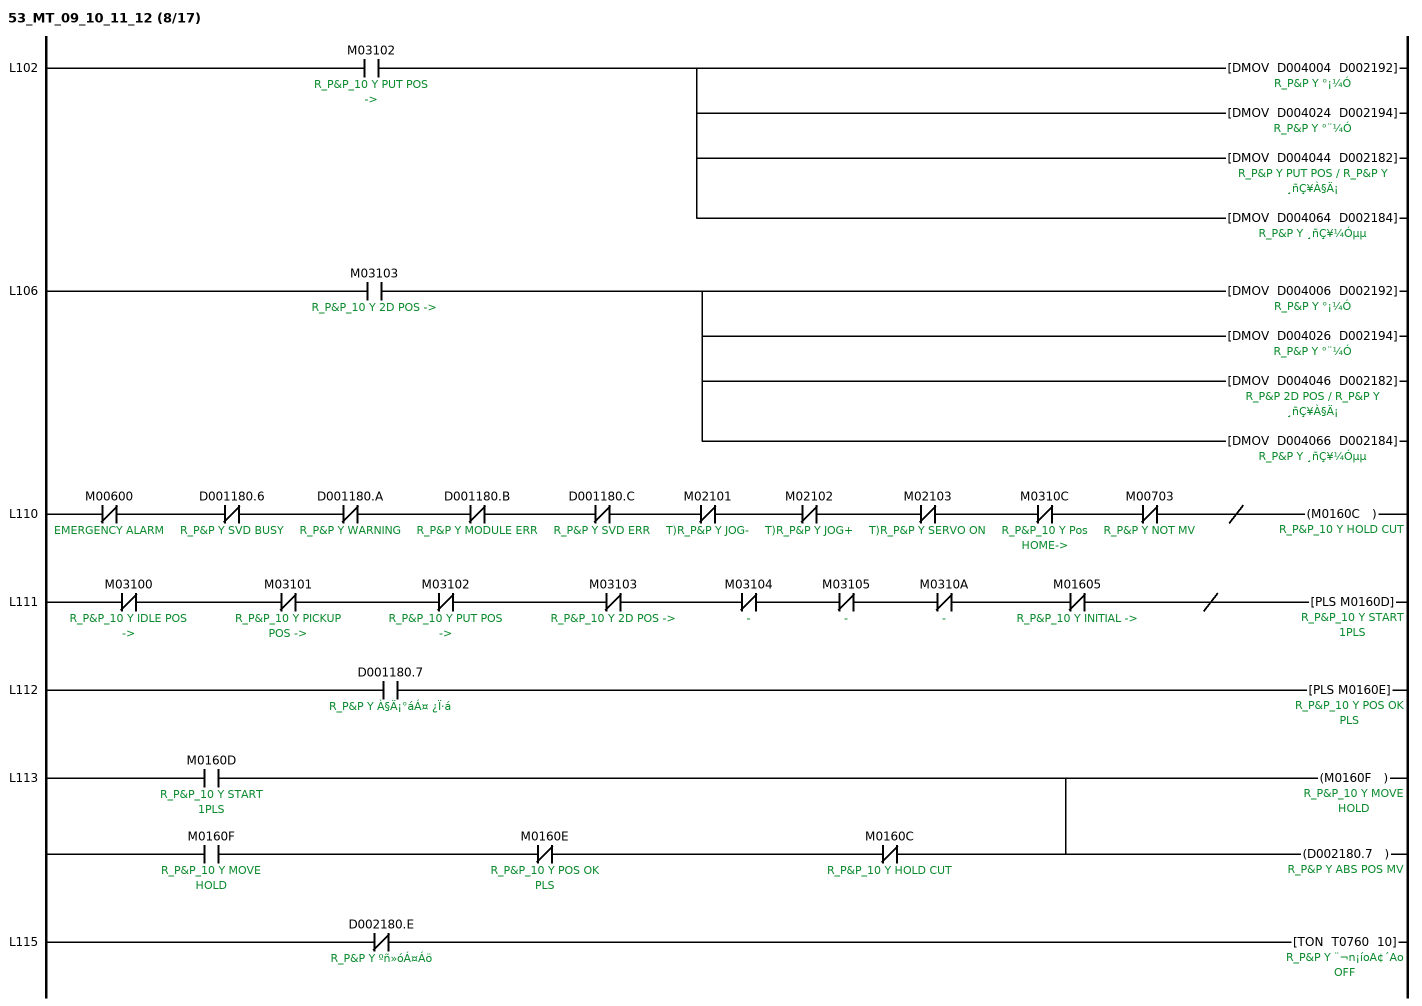
; L102
LOAD      M03102	// R_P&P_10 Y PUT POS ->
DMOV      D004004 D002192	// R_P&P Y °¡¼Ó
DMOV      D004024 D002194	// R_P&P Y °¨¼Ó
DMOV      D004044 D002182	// R_P&P Y PUT POS / R_P&P Y ¸ñÇ¥À§Ä¡
DMOV      D004064 D002184	// R_P&P Y ¸ñÇ¥¼Óµµ
; L106
LOAD      M03103	// R_P&P_10 Y 2D POS ->
DMOV      D004006 D002192	// R_P&P Y °¡¼Ó
DMOV      D004026 D002194	// R_P&P Y °¨¼Ó
DMOV      D004046 D002182	// R_P&P 2D POS / R_P&P Y ¸ñÇ¥À§Ä¡
DMOV      D004066 D002184	// R_P&P Y ¸ñÇ¥¼Óµµ
; L110
LOAD NOT  M00600	// EMERGENCY ALARM
AND NOT   D001180.6	// R_P&P Y SVD BUSY
AND NOT   D001180.A	// R_P&P Y WARNING
AND NOT   D001180.B	// R_P&P Y MODULE ERR
AND NOT   D001180.C	// R_P&P Y SVD ERR
AND NOT   M02101	// T)R_P&P Y JOG-
AND NOT   M02102	// T)R_P&P Y JOG+
AND NOT   M02103	// T)R_P&P Y SERVO ON
AND NOT   M0310C	// R_P&P_10 Y Pos HOME->
AND NOT   M00703	// R_P&P Y NOT MV
NOT
OUT       M0160C	// R_P&P_10 Y HOLD CUT
; L111
LOAD NOT  M03100	// R_P&P_10 Y IDLE POS ->
AND NOT   M03101	// R_P&P_10 Y PICKUP POS ->
AND NOT   M03102	// R_P&P_10 Y PUT POS ->
AND NOT   M03103	// R_P&P_10 Y 2D POS ->
AND NOT   M03104	// -
AND NOT   M03105	// -
AND NOT   M0310A	// -
AND NOT   M01605	// R_P&P_10 Y INITIAL ->
NOT
OUTP      M0160D	// R_P&P_10 Y START 1PLS
; L112
LOAD      D001180.7	// R_P&P Y À§Ä¡°áÁ¤ ¿Ï·á
OUTP      M0160E	// R_P&P_10 Y POS OK PLS
; L113
LOAD      M0160D	// R_P&P_10 Y START 1PLS
LOAD      M0160F	// R_P&P_10 Y MOVE HOLD
AND NOT   M0160E	// R_P&P_10 Y POS OK PLS
AND NOT   M0160C	// R_P&P_10 Y HOLD CUT
OR LOAD
OUT       M0160F	// R_P&P_10 Y MOVE HOLD
OUT       D002180.7	// R_P&P Y ABS POS MV
; L115
LOAD NOT  D002180.E	// R_P&P Y ºñ»óÁ¤Áö
TON       T0760 10	// R_P&P Y ¨¬n¡íoA¢´AoOFF

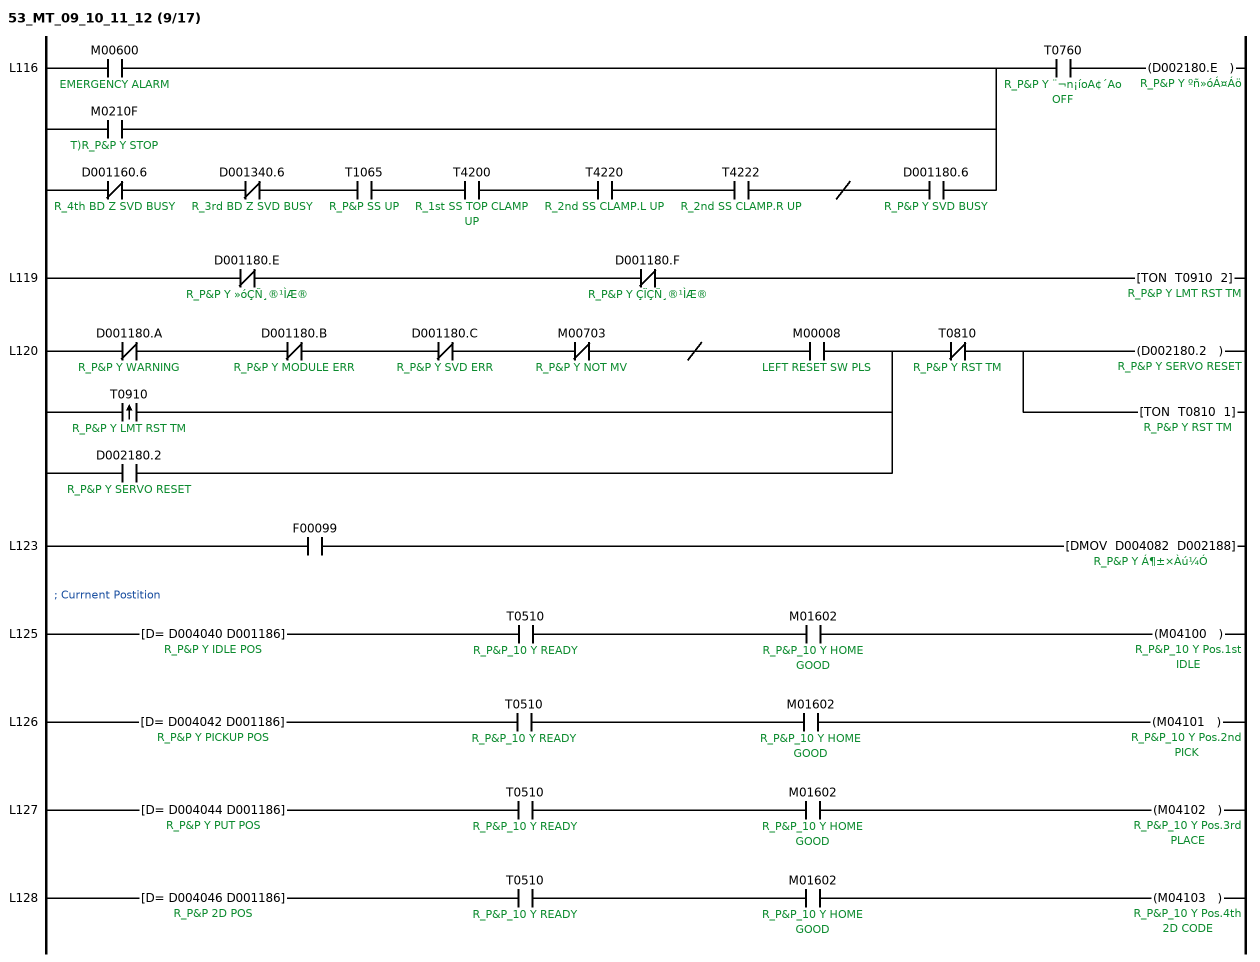
; L116
LOAD      M00600	// EMERGENCY ALARM
OR        M0210F	// T)R_P&P Y STOP
LOAD NOT  D001160.6	// R_4th BD Z SVD BUSY
AND NOT   D001340.6	// R_3rd BD Z SVD BUSY
AND       T1065	// R_P&P SS UP
AND       T4200	// R_1st SS TOP CLAMP UP
AND       T4220	// R_2nd SS CLAMP.L UP
AND       T4222	// R_2nd SS CLAMP.R UP
NOT
AND       D001180.6	// R_P&P Y SVD BUSY
OR LOAD
AND       T0760	// R_P&P Y ¨¬n¡íoA¢´AoOFF
OUT       D002180.E	// R_P&P Y ºñ»óÁ¤Áö
; L119
LOAD NOT  D001180.E	// R_P&P Y »óÇÑ¸®¹ÌÆ®
AND NOT   D001180.F	// R_P&P Y ÇÏÇÑ¸®¹ÌÆ®
TON       T0910 2	// R_P&P Y LMT RST TM
; L120
LOAD NOT  D001180.A	// R_P&P Y WARNING
AND NOT   D001180.B	// R_P&P Y MODULE ERR
AND NOT   D001180.C	// R_P&P Y SVD ERR
AND NOT   M00703	// R_P&P Y NOT MV
NOT
AND       M00008	// LEFT RESET SW PLS
ORP       T0910	// R_P&P Y LMT RST TM
OR        D002180.2	// R_P&P Y SERVO RESET
AND NOT   T0810	// R_P&P Y RST TM
OUT       D002180.2	// R_P&P Y SERVO RESET
TON       T0810 1	// R_P&P Y RST TM
; L123
LOAD      F00099
DMOV      D004082 D002188	// R_P&P Y Á¶±×Àú¼Ó
// Currnent Postition
; L125
LOADD=    D004040 D001186	// R_P&P Y IDLE POS
AND       T0510	// R_P&P_10 Y READY
AND       M01602	// R_P&P_10 Y HOME GOOD
OUT       M04100	// R_P&P_10 Y Pos.1st IDLE
; L126
LOADD=    D004042 D001186	// R_P&P Y PICKUP POS
AND       T0510	// R_P&P_10 Y READY
AND       M01602	// R_P&P_10 Y HOME GOOD
OUT       M04101	// R_P&P_10 Y Pos.2nd PICK
; L127
LOADD=    D004044 D001186	// R_P&P Y PUT POS
AND       T0510	// R_P&P_10 Y READY
AND       M01602	// R_P&P_10 Y HOME GOOD
OUT       M04102	// R_P&P_10 Y Pos.3rd PLACE
; L128
LOADD=    D004046 D001186	// R_P&P 2D POS
AND       T0510	// R_P&P_10 Y READY
AND       M01602	// R_P&P_10 Y HOME GOOD
OUT       M04103	// R_P&P_10 Y Pos.4th 2D CODE

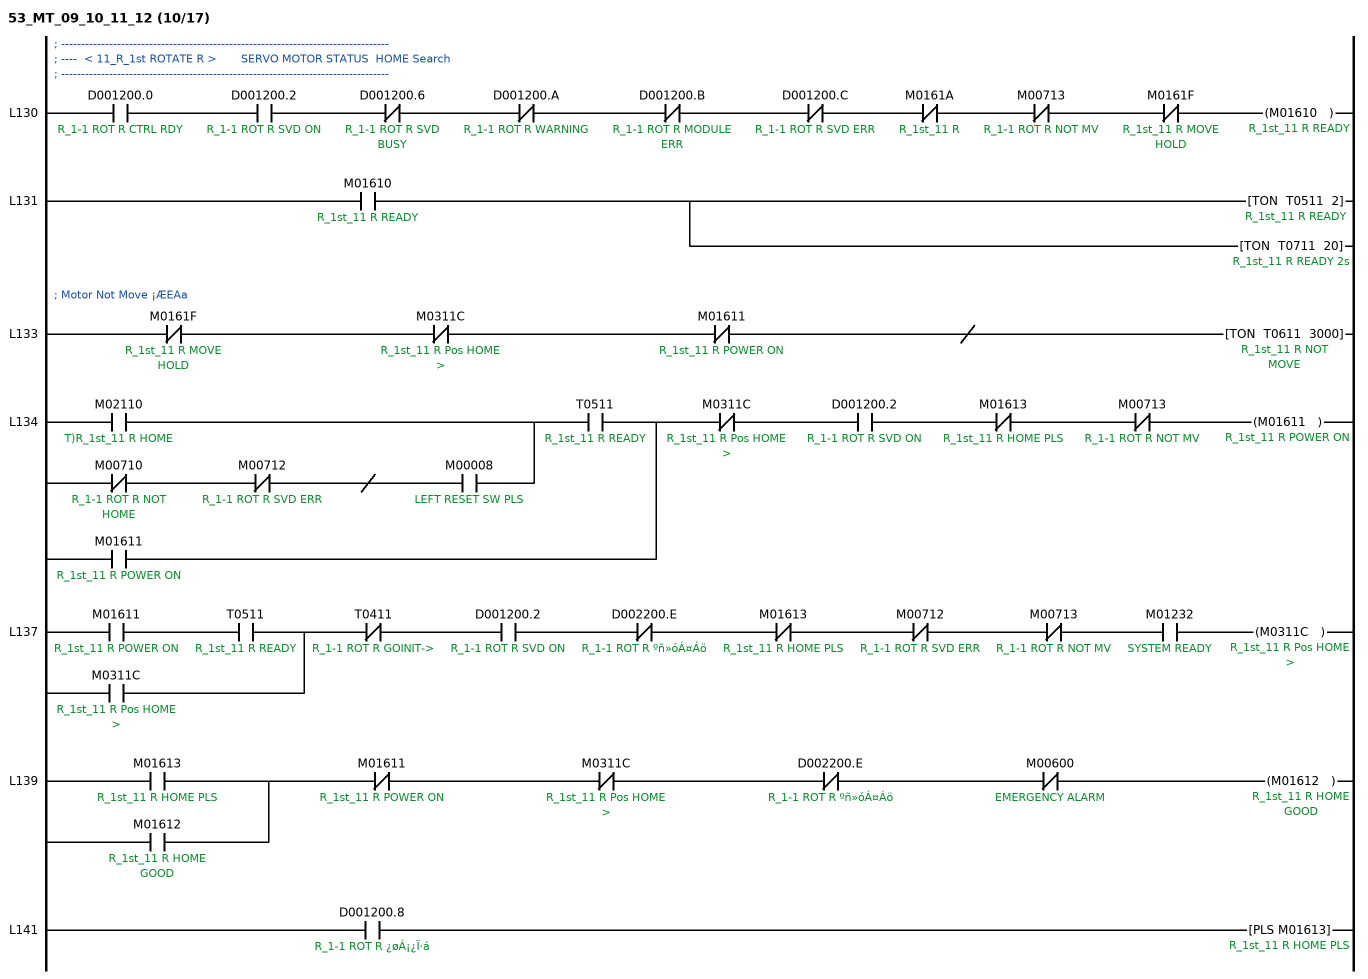
// ----------------------------------------------------------------------------------
// 
// ----  < 11_R_1st ROTATE R >       SERVO MOTOR STATUS  HOME Search
// 
// ----------------------------------------------------------------------------------
; L130
LOAD      D001200.0	// R_1-1 ROT R CTRL RDY
AND       D001200.2	// R_1-1 ROT R SVD ON
AND NOT   D001200.6	// R_1-1 ROT R SVD BUSY
AND NOT   D001200.A	// R_1-1 ROT R WARNING
AND NOT   D001200.B	// R_1-1 ROT R MODULE ERR
AND NOT   D001200.C	// R_1-1 ROT R SVD ERR
AND NOT   M0161A	// R_1st_11 R
AND NOT   M00713	// R_1-1 ROT R NOT MV
AND NOT   M0161F	// R_1st_11 R MOVE HOLD
OUT       M01610	// R_1st_11 R READY
; L131
LOAD      M01610	// R_1st_11 R READY
TON       T0511 2	// R_1st_11 R READY
TON       T0711 20	// R_1st_11 R READY 2s
; L133
LOAD NOT  M0161F	// R_1st_11 R MOVE HOLD
AND NOT   M0311C	// R_1st_11 R Pos HOME >
AND NOT   M01611	// R_1st_11 R POWER ON
NOT
TON       T0611 3000	// R_1st_11 R NOT MOVE
// output comment: Motor Not Move ¡ÆEAa
; L134
LOAD      M02110	// T)R_1st_11 R HOME
LOAD NOT  M00710	// R_1-1 ROT R NOT HOME
AND NOT   M00712	// R_1-1 ROT R SVD ERR
NOT
AND       M00008	// LEFT RESET SW PLS
OR LOAD
AND       T0511	// R_1st_11 R READY
OR        M01611	// R_1st_11 R POWER ON
AND NOT   M0311C	// R_1st_11 R Pos HOME >
AND       D001200.2	// R_1-1 ROT R SVD ON
AND NOT   M01613	// R_1st_11 R HOME PLS
AND NOT   M00713	// R_1-1 ROT R NOT MV
OUT       M01611	// R_1st_11 R POWER ON
; L137
LOAD      M01611	// R_1st_11 R POWER ON
AND       T0511	// R_1st_11 R READY
OR        M0311C	// R_1st_11 R Pos HOME >
AND NOT   T0411	// R_1-1 ROT R GOINIT->
AND       D001200.2	// R_1-1 ROT R SVD ON
AND NOT   D002200.E	// R_1-1 ROT R ºñ»óÁ¤Áö
AND NOT   M01613	// R_1st_11 R HOME PLS
AND NOT   M00712	// R_1-1 ROT R SVD ERR
AND NOT   M00713	// R_1-1 ROT R NOT MV
AND       M01232	// SYSTEM READY
OUT       M0311C	// R_1st_11 R Pos HOME >
; L139
LOAD      M01613	// R_1st_11 R HOME PLS
OR        M01612	// R_1st_11 R HOME GOOD
AND NOT   M01611	// R_1st_11 R POWER ON
AND NOT   M0311C	// R_1st_11 R Pos HOME >
AND NOT   D002200.E	// R_1-1 ROT R ºñ»óÁ¤Áö
AND NOT   M00600	// EMERGENCY ALARM
OUT       M01612	// R_1st_11 R HOME GOOD
; L141
LOAD      D001200.8	// R_1-1 ROT R ¿øÁ¡¿Ï·á
OUTP      M01613	// R_1st_11 R HOME PLS

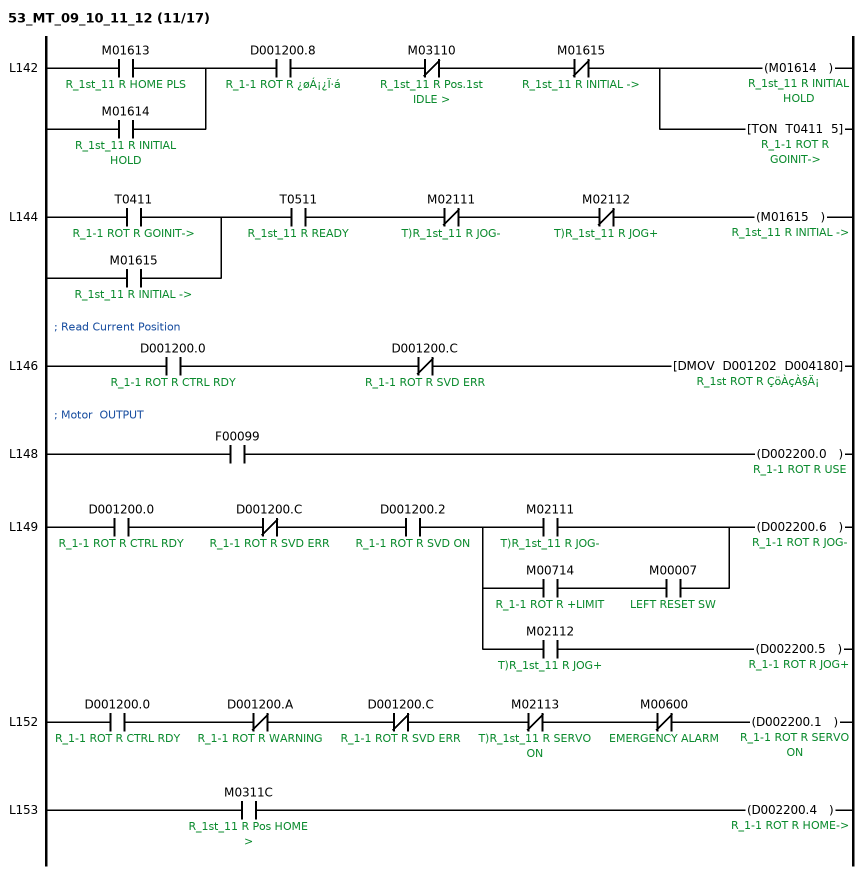
; L142
LOAD      M01613	// R_1st_11 R HOME PLS
OR        M01614	// R_1st_11 R INITIAL HOLD
AND       D001200.8	// R_1-1 ROT R ¿øÁ¡¿Ï·á
AND NOT   M03110	// R_1st_11 R Pos.1st IDLE >
AND NOT   M01615	// R_1st_11 R INITIAL ->
OUT       M01614	// R_1st_11 R INITIAL HOLD
TON       T0411 5	// R_1-1 ROT R GOINIT->
; L144
LOAD      T0411	// R_1-1 ROT R GOINIT->
OR        M01615	// R_1st_11 R INITIAL ->
AND       T0511	// R_1st_11 R READY
AND NOT   M02111	// T)R_1st_11 R JOG-
AND NOT   M02112	// T)R_1st_11 R JOG+
OUT       M01615	// R_1st_11 R INITIAL ->
; L146
LOAD      D001200.0	// R_1-1 ROT R CTRL RDY
AND NOT   D001200.C	// R_1-1 ROT R SVD ERR
DMOV      D001202 D004180	// R_1st ROT R ÇöÀçÀ§Ä¡
// output comment: Read Current Position
//  Motor  OUTPUT
; L148
LOAD      F00099
OUT       D002200.0	// R_1-1 ROT R USE
; L149
LOAD      D001200.0	// R_1-1 ROT R CTRL RDY
AND NOT   D001200.C	// R_1-1 ROT R SVD ERR
AND       D001200.2	// R_1-1 ROT R SVD ON
MPUSH
LOAD      M02111	// T)R_1st_11 R JOG-
LOAD      M00714	// R_1-1 ROT R +LIMIT
AND       M00007	// LEFT RESET SW
OR LOAD
AND LOAD
OUT       D002200.6	// R_1-1 ROT R JOG-
MPOP
AND       M02112	// T)R_1st_11 R JOG+
OUT       D002200.5	// R_1-1 ROT R JOG+
; L152
LOAD      D001200.0	// R_1-1 ROT R CTRL RDY
AND NOT   D001200.A	// R_1-1 ROT R WARNING
AND NOT   D001200.C	// R_1-1 ROT R SVD ERR
AND NOT   M02113	// T)R_1st_11 R SERVO ON
AND NOT   M00600	// EMERGENCY ALARM
OUT       D002200.1	// R_1-1 ROT R SERVO ON
; L153
LOAD      M0311C	// R_1st_11 R Pos HOME >
OUT       D002200.4	// R_1-1 ROT R HOME->

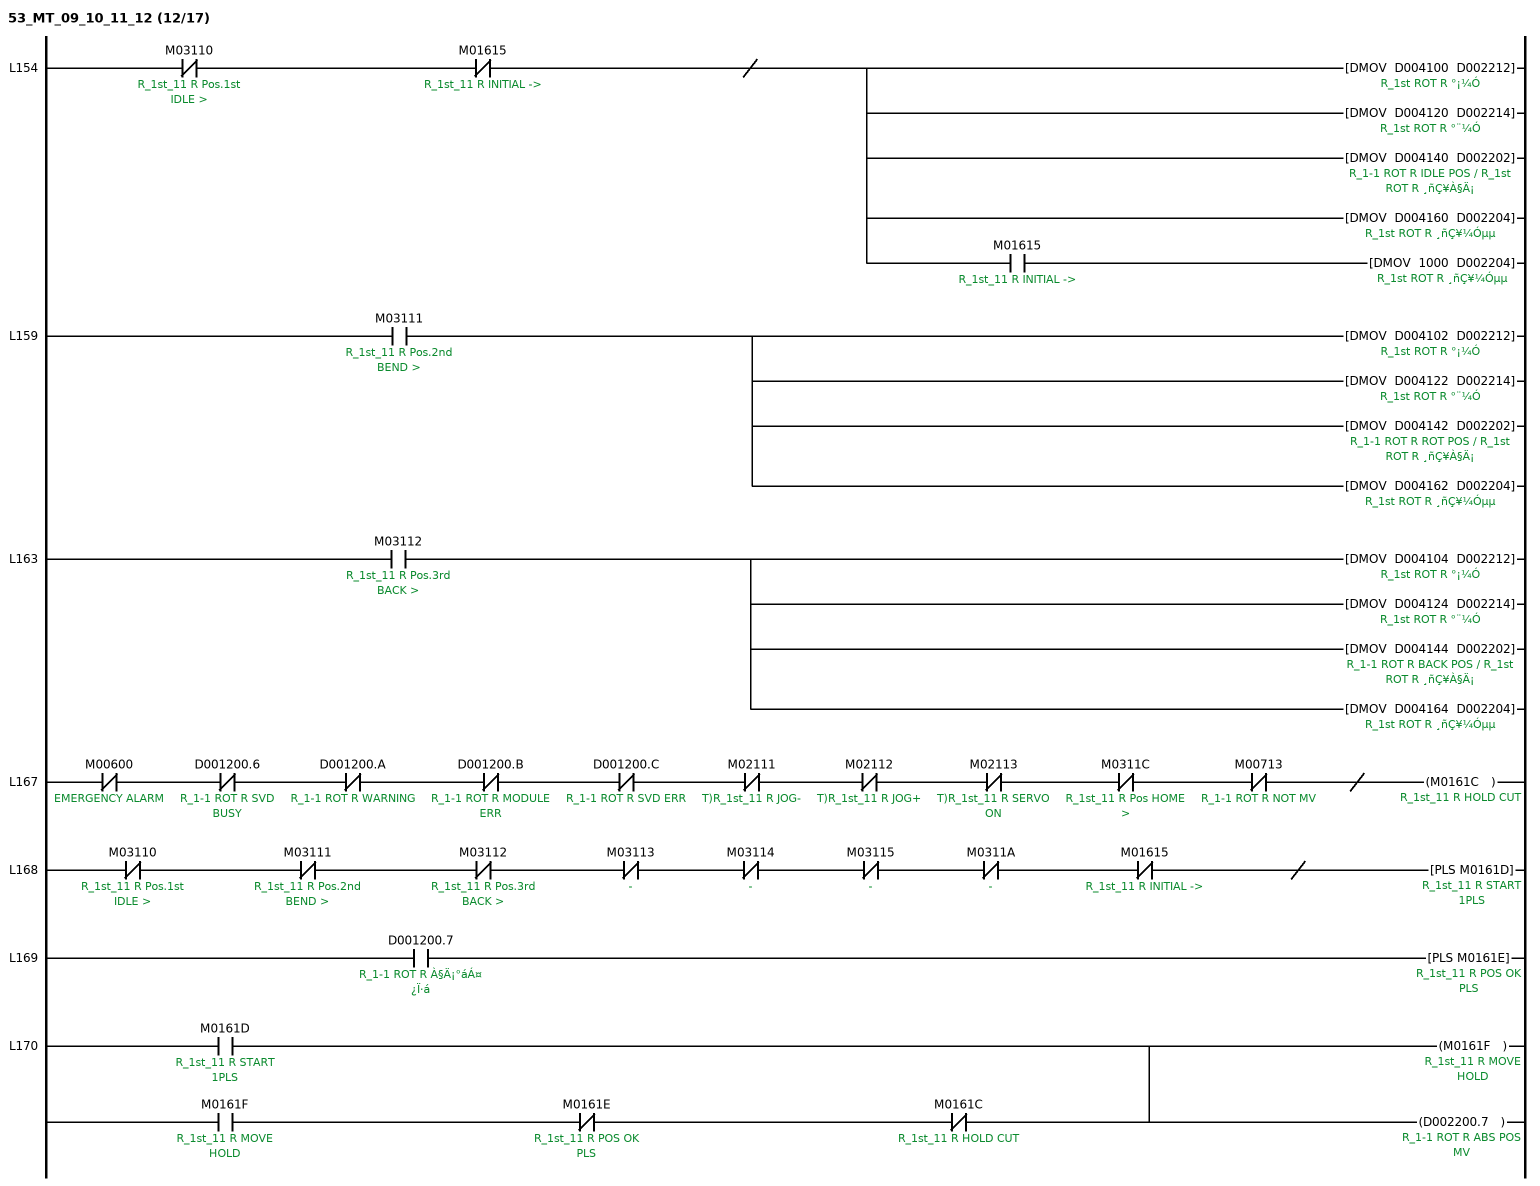
; L154
LOAD NOT  M03110	// R_1st_11 R Pos.1st IDLE >
AND NOT   M01615	// R_1st_11 R INITIAL ->
NOT
DMOV      D004100 D002212	// R_1st ROT R °¡¼Ó
DMOV      D004120 D002214	// R_1st ROT R °¨¼Ó
DMOV      D004140 D002202	// R_1-1 ROT R IDLE POS / R_1st ROT R ¸ñÇ¥À§Ä¡
DMOV      D004160 D002204	// R_1st ROT R ¸ñÇ¥¼Óµµ
AND       M01615	// R_1st_11 R INITIAL ->
DMOV      1000 D002204	// R_1st ROT R ¸ñÇ¥¼Óµµ
; L159
LOAD      M03111	// R_1st_11 R Pos.2nd BEND >
DMOV      D004102 D002212	// R_1st ROT R °¡¼Ó
DMOV      D004122 D002214	// R_1st ROT R °¨¼Ó
DMOV      D004142 D002202	// R_1-1 ROT R ROT POS / R_1st ROT R ¸ñÇ¥À§Ä¡
DMOV      D004162 D002204	// R_1st ROT R ¸ñÇ¥¼Óµµ
; L163
LOAD      M03112	// R_1st_11 R Pos.3rd BACK >
DMOV      D004104 D002212	// R_1st ROT R °¡¼Ó
DMOV      D004124 D002214	// R_1st ROT R °¨¼Ó
DMOV      D004144 D002202	// R_1-1 ROT R BACK POS / R_1st ROT R ¸ñÇ¥À§Ä¡
DMOV      D004164 D002204	// R_1st ROT R ¸ñÇ¥¼Óµµ
; L167
LOAD NOT  M00600	// EMERGENCY ALARM
AND NOT   D001200.6	// R_1-1 ROT R SVD BUSY
AND NOT   D001200.A	// R_1-1 ROT R WARNING
AND NOT   D001200.B	// R_1-1 ROT R MODULE ERR
AND NOT   D001200.C	// R_1-1 ROT R SVD ERR
AND NOT   M02111	// T)R_1st_11 R JOG-
AND NOT   M02112	// T)R_1st_11 R JOG+
AND NOT   M02113	// T)R_1st_11 R SERVO ON
AND NOT   M0311C	// R_1st_11 R Pos HOME >
AND NOT   M00713	// R_1-1 ROT R NOT MV
NOT
OUT       M0161C	// R_1st_11 R HOLD CUT
; L168
LOAD NOT  M03110	// R_1st_11 R Pos.1st IDLE >
AND NOT   M03111	// R_1st_11 R Pos.2nd BEND >
AND NOT   M03112	// R_1st_11 R Pos.3rd BACK >
AND NOT   M03113	// -
AND NOT   M03114	// -
AND NOT   M03115	// -
AND NOT   M0311A	// -
AND NOT   M01615	// R_1st_11 R INITIAL ->
NOT
OUTP      M0161D	// R_1st_11 R START 1PLS
; L169
LOAD      D001200.7	// R_1-1 ROT R À§Ä¡°áÁ¤ ¿Ï·á
OUTP      M0161E	// R_1st_11 R POS OK PLS
; L170
LOAD      M0161D	// R_1st_11 R START 1PLS
LOAD      M0161F	// R_1st_11 R MOVE HOLD
AND NOT   M0161E	// R_1st_11 R POS OK PLS
AND NOT   M0161C	// R_1st_11 R HOLD CUT
OR LOAD
OUT       M0161F	// R_1st_11 R MOVE HOLD
OUT       D002200.7	// R_1-1 ROT R ABS POS MV

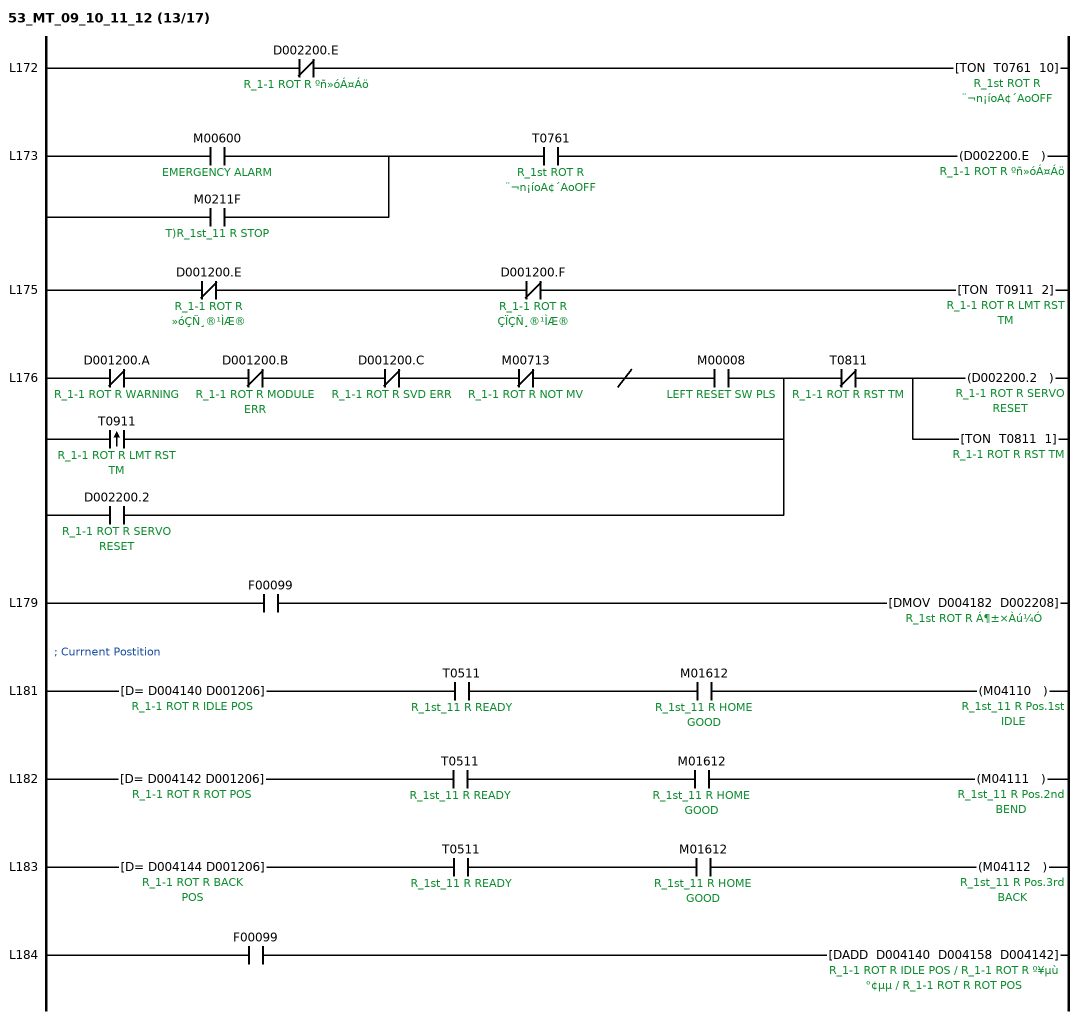
; L172
LOAD NOT  D002200.E	// R_1-1 ROT R ºñ»óÁ¤Áö
TON       T0761 10	// R_1st ROT R ¨¬n¡íoA¢´AoOFF
; L173
LOAD      M00600	// EMERGENCY ALARM
OR        M0211F	// T)R_1st_11 R STOP
AND       T0761	// R_1st ROT R ¨¬n¡íoA¢´AoOFF
OUT       D002200.E	// R_1-1 ROT R ºñ»óÁ¤Áö
; L175
LOAD NOT  D001200.E	// R_1-1 ROT R »óÇÑ¸®¹ÌÆ®
AND NOT   D001200.F	// R_1-1 ROT R ÇÏÇÑ¸®¹ÌÆ®
TON       T0911 2	// R_1-1 ROT R LMT RST TM
; L176
LOAD NOT  D001200.A	// R_1-1 ROT R WARNING
AND NOT   D001200.B	// R_1-1 ROT R MODULE ERR
AND NOT   D001200.C	// R_1-1 ROT R SVD ERR
AND NOT   M00713	// R_1-1 ROT R NOT MV
NOT
AND       M00008	// LEFT RESET SW PLS
ORP       T0911	// R_1-1 ROT R LMT RST TM
OR        D002200.2	// R_1-1 ROT R SERVO RESET
AND NOT   T0811	// R_1-1 ROT R RST TM
OUT       D002200.2	// R_1-1 ROT R SERVO RESET
TON       T0811 1	// R_1-1 ROT R RST TM
; L179
LOAD      F00099
DMOV      D004182 D002208	// R_1st ROT R Á¶±×Àú¼Ó
// Currnent Postition
; L181
LOADD=    D004140 D001206	// R_1-1 ROT R IDLE POS
AND       T0511	// R_1st_11 R READY
AND       M01612	// R_1st_11 R HOME GOOD
OUT       M04110	// R_1st_11 R Pos.1st IDLE
; L182
LOADD=    D004142 D001206	// R_1-1 ROT R ROT POS
AND       T0511	// R_1st_11 R READY
AND       M01612	// R_1st_11 R HOME GOOD
OUT       M04111	// R_1st_11 R Pos.2nd BEND
; L183
LOADD=    D004144 D001206	// R_1-1 ROT R BACK POS
AND       T0511	// R_1st_11 R READY
AND       M01612	// R_1st_11 R HOME GOOD
OUT       M04112	// R_1st_11 R Pos.3rd BACK
; L184
LOAD      F00099
DADD      D004140 D004158 D004142	// R_1-1 ROT R IDLE POS / R_1-1 ROT R º¥µù °¢µµ / R_1-1 ROT R ROT POS

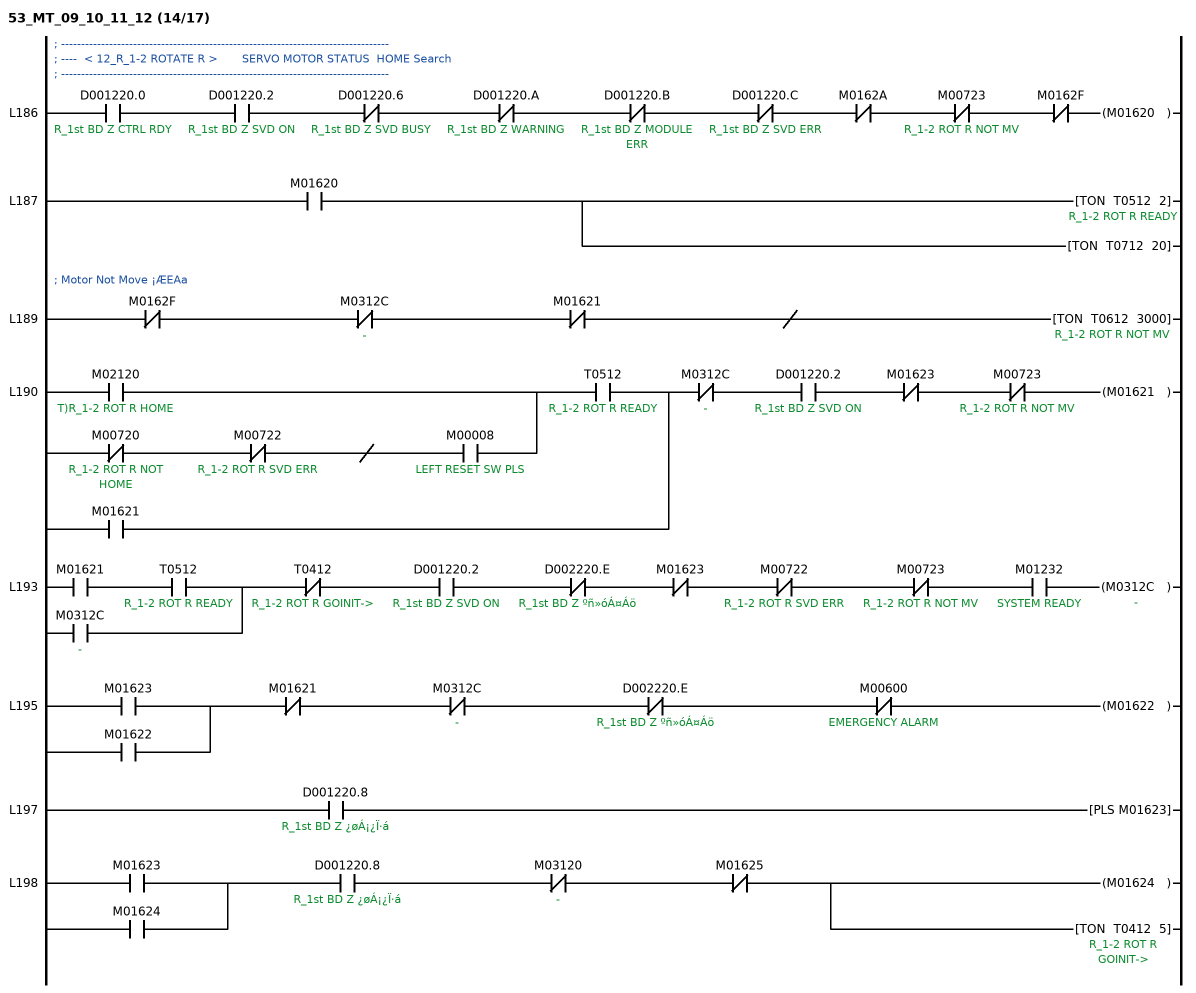
// ----------------------------------------------------------------------------------
// 
// ----  < 12_R_1-2 ROTATE R >       SERVO MOTOR STATUS  HOME Search
// 
// ----------------------------------------------------------------------------------
; L186
LOAD      D001220.0	// R_1st BD Z CTRL RDY
AND       D001220.2	// R_1st BD Z SVD ON
AND NOT   D001220.6	// R_1st BD Z SVD BUSY
AND NOT   D001220.A	// R_1st BD Z WARNING
AND NOT   D001220.B	// R_1st BD Z MODULE ERR
AND NOT   D001220.C	// R_1st BD Z SVD ERR
AND NOT   M0162A
AND NOT   M00723	// R_1-2 ROT R NOT MV
AND NOT   M0162F
OUT       M01620
; L187
LOAD      M01620
TON       T0512 2	// R_1-2 ROT R READY
TON       T0712 20
; L189
LOAD NOT  M0162F
AND NOT   M0312C	// -
AND NOT   M01621
NOT
TON       T0612 3000	// R_1-2 ROT R NOT MV
// output comment: Motor Not Move ¡ÆEAa
; L190
LOAD      M02120	// T)R_1-2 ROT R HOME
LOAD NOT  M00720	// R_1-2 ROT R NOT HOME
AND NOT   M00722	// R_1-2 ROT R SVD ERR
NOT
AND       M00008	// LEFT RESET SW PLS
OR LOAD
AND       T0512	// R_1-2 ROT R READY
OR        M01621
AND NOT   M0312C	// -
AND       D001220.2	// R_1st BD Z SVD ON
AND NOT   M01623
AND NOT   M00723	// R_1-2 ROT R NOT MV
OUT       M01621
; L193
LOAD      M01621
AND       T0512	// R_1-2 ROT R READY
OR        M0312C	// -
AND NOT   T0412	// R_1-2 ROT R GOINIT->
AND       D001220.2	// R_1st BD Z SVD ON
AND NOT   D002220.E	// R_1st BD Z ºñ»óÁ¤Áö
AND NOT   M01623
AND NOT   M00722	// R_1-2 ROT R SVD ERR
AND NOT   M00723	// R_1-2 ROT R NOT MV
AND       M01232	// SYSTEM READY
OUT       M0312C	// -
; L195
LOAD      M01623
OR        M01622
AND NOT   M01621
AND NOT   M0312C	// -
AND NOT   D002220.E	// R_1st BD Z ºñ»óÁ¤Áö
AND NOT   M00600	// EMERGENCY ALARM
OUT       M01622
; L197
LOAD      D001220.8	// R_1st BD Z ¿øÁ¡¿Ï·á
OUTP      M01623
; L198
LOAD      M01623
OR        M01624
AND       D001220.8	// R_1st BD Z ¿øÁ¡¿Ï·á
AND NOT   M03120	// -
AND NOT   M01625
OUT       M01624
TON       T0412 5	// R_1-2 ROT R GOINIT->

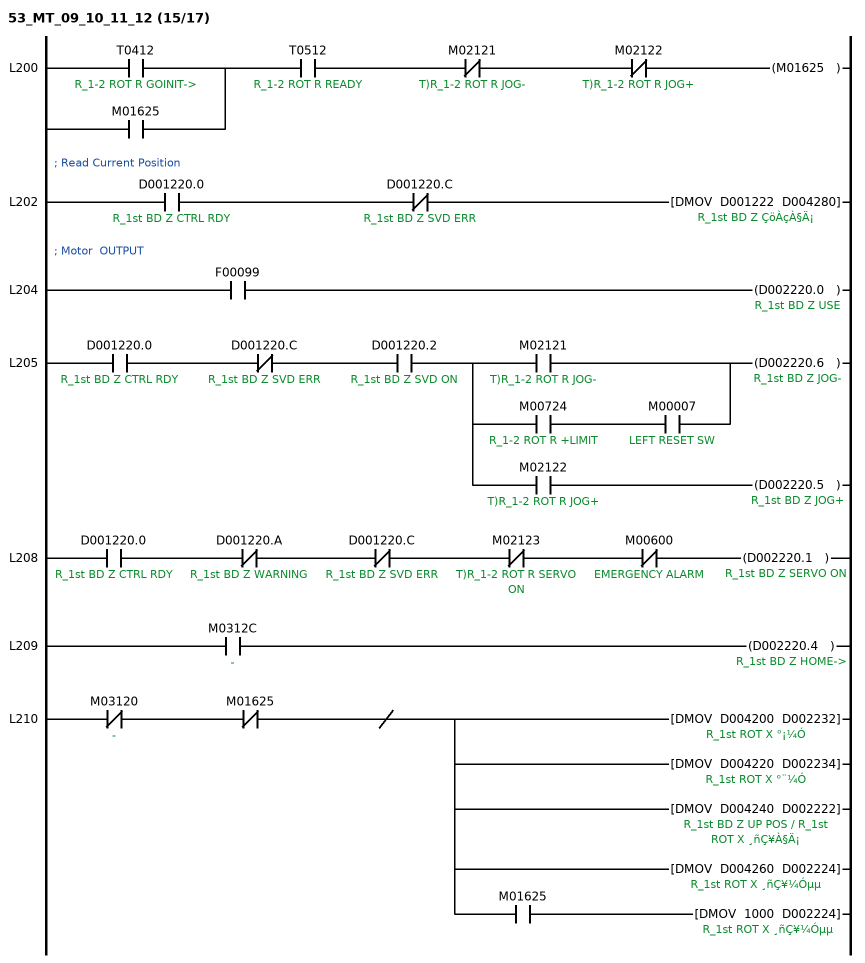
; L200
LOAD      T0412	// R_1-2 ROT R GOINIT->
OR        M01625
AND       T0512	// R_1-2 ROT R READY
AND NOT   M02121	// T)R_1-2 ROT R JOG-
AND NOT   M02122	// T)R_1-2 ROT R JOG+
OUT       M01625
; L202
LOAD      D001220.0	// R_1st BD Z CTRL RDY
AND NOT   D001220.C	// R_1st BD Z SVD ERR
DMOV      D001222 D004280	// R_1st BD Z ÇöÀçÀ§Ä¡
// output comment: Read Current Position
//  Motor  OUTPUT
; L204
LOAD      F00099
OUT       D002220.0	// R_1st BD Z USE
; L205
LOAD      D001220.0	// R_1st BD Z CTRL RDY
AND NOT   D001220.C	// R_1st BD Z SVD ERR
AND       D001220.2	// R_1st BD Z SVD ON
MPUSH
LOAD      M02121	// T)R_1-2 ROT R JOG-
LOAD      M00724	// R_1-2 ROT R +LIMIT
AND       M00007	// LEFT RESET SW
OR LOAD
AND LOAD
OUT       D002220.6	// R_1st BD Z JOG-
MPOP
AND       M02122	// T)R_1-2 ROT R JOG+
OUT       D002220.5	// R_1st BD Z JOG+
; L208
LOAD      D001220.0	// R_1st BD Z CTRL RDY
AND NOT   D001220.A	// R_1st BD Z WARNING
AND NOT   D001220.C	// R_1st BD Z SVD ERR
AND NOT   M02123	// T)R_1-2 ROT R SERVO ON
AND NOT   M00600	// EMERGENCY ALARM
OUT       D002220.1	// R_1st BD Z SERVO ON
; L209
LOAD      M0312C	// -
OUT       D002220.4	// R_1st BD Z HOME->
; L210
LOAD NOT  M03120	// -
AND NOT   M01625
NOT
DMOV      D004200 D002232	// R_1st ROT X °¡¼Ó
DMOV      D004220 D002234	// R_1st ROT X °¨¼Ó
DMOV      D004240 D002222	// R_1st BD Z UP POS / R_1st ROT X ¸ñÇ¥À§Ä¡
DMOV      D004260 D002224	// R_1st ROT X ¸ñÇ¥¼Óµµ
AND       M01625
DMOV      1000 D002224	// R_1st ROT X ¸ñÇ¥¼Óµµ

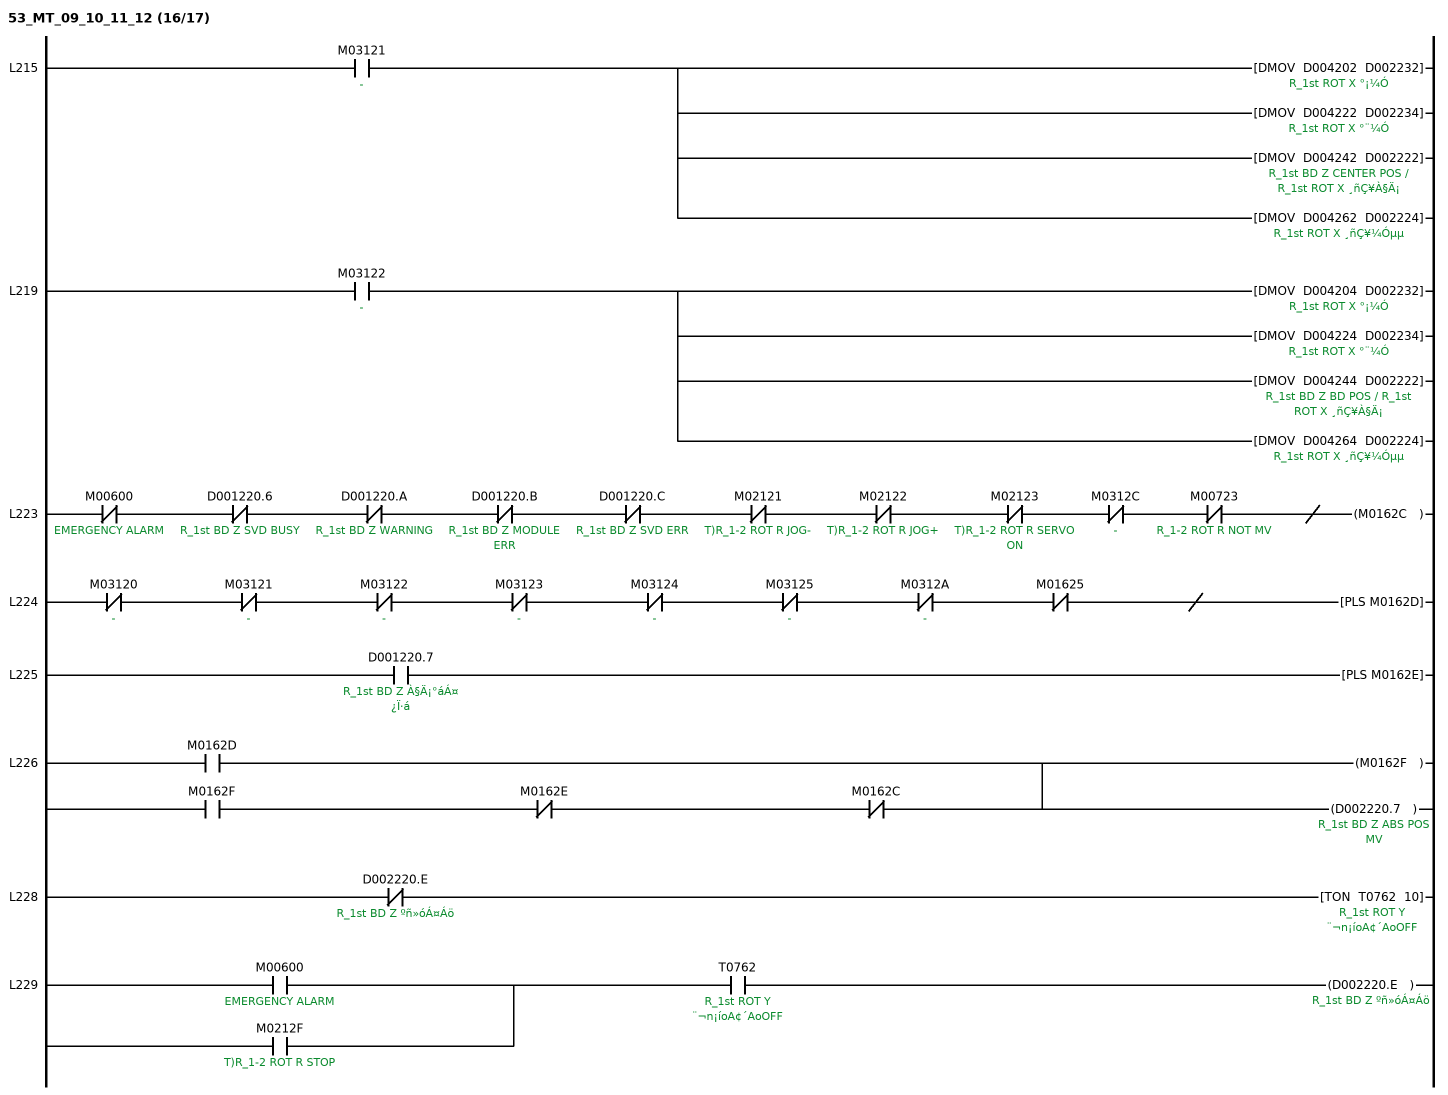
; L215
LOAD      M03121	// -
DMOV      D004202 D002232	// R_1st ROT X °¡¼Ó
DMOV      D004222 D002234	// R_1st ROT X °¨¼Ó
DMOV      D004242 D002222	// R_1st BD Z CENTER POS / R_1st ROT X ¸ñÇ¥À§Ä¡
DMOV      D004262 D002224	// R_1st ROT X ¸ñÇ¥¼Óµµ
; L219
LOAD      M03122	// -
DMOV      D004204 D002232	// R_1st ROT X °¡¼Ó
DMOV      D004224 D002234	// R_1st ROT X °¨¼Ó
DMOV      D004244 D002222	// R_1st BD Z BD POS / R_1st ROT X ¸ñÇ¥À§Ä¡
DMOV      D004264 D002224	// R_1st ROT X ¸ñÇ¥¼Óµµ
; L223
LOAD NOT  M00600	// EMERGENCY ALARM
AND NOT   D001220.6	// R_1st BD Z SVD BUSY
AND NOT   D001220.A	// R_1st BD Z WARNING
AND NOT   D001220.B	// R_1st BD Z MODULE ERR
AND NOT   D001220.C	// R_1st BD Z SVD ERR
AND NOT   M02121	// T)R_1-2 ROT R JOG-
AND NOT   M02122	// T)R_1-2 ROT R JOG+
AND NOT   M02123	// T)R_1-2 ROT R SERVO ON
AND NOT   M0312C	// -
AND NOT   M00723	// R_1-2 ROT R NOT MV
NOT
OUT       M0162C
; L224
LOAD NOT  M03120	// -
AND NOT   M03121	// -
AND NOT   M03122	// -
AND NOT   M03123	// -
AND NOT   M03124	// -
AND NOT   M03125	// -
AND NOT   M0312A	// -
AND NOT   M01625
NOT
OUTP      M0162D
; L225
LOAD      D001220.7	// R_1st BD Z À§Ä¡°áÁ¤ ¿Ï·á
OUTP      M0162E
; L226
LOAD      M0162D
LOAD      M0162F
AND NOT   M0162E
AND NOT   M0162C
OR LOAD
OUT       M0162F
OUT       D002220.7	// R_1st BD Z ABS POS MV
; L228
LOAD NOT  D002220.E	// R_1st BD Z ºñ»óÁ¤Áö
TON       T0762 10	// R_1st ROT Y ¨¬n¡íoA¢´AoOFF
; L229
LOAD      M00600	// EMERGENCY ALARM
OR        M0212F	// T)R_1-2 ROT R STOP
AND       T0762	// R_1st ROT Y ¨¬n¡íoA¢´AoOFF
OUT       D002220.E	// R_1st BD Z ºñ»óÁ¤Áö

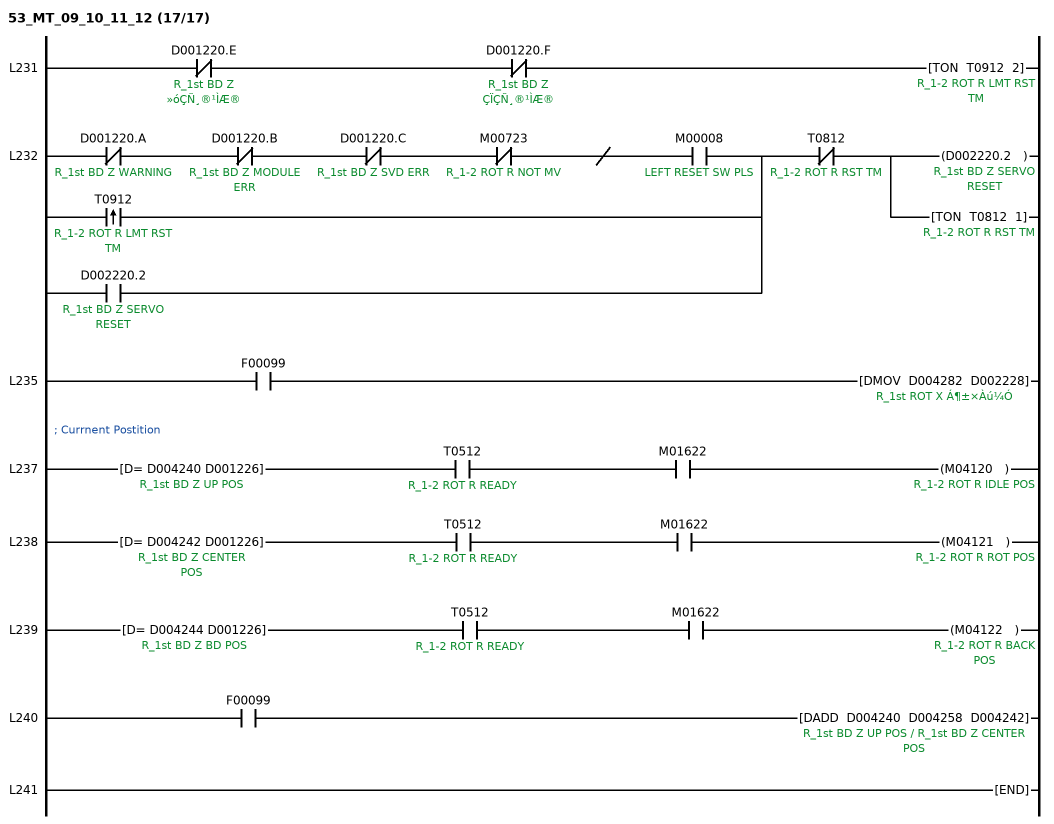
; L231
LOAD NOT  D001220.E	// R_1st BD Z »óÇÑ¸®¹ÌÆ®
AND NOT   D001220.F	// R_1st BD Z ÇÏÇÑ¸®¹ÌÆ®
TON       T0912 2	// R_1-2 ROT R LMT RST TM
; L232
LOAD NOT  D001220.A	// R_1st BD Z WARNING
AND NOT   D001220.B	// R_1st BD Z MODULE ERR
AND NOT   D001220.C	// R_1st BD Z SVD ERR
AND NOT   M00723	// R_1-2 ROT R NOT MV
NOT
AND       M00008	// LEFT RESET SW PLS
ORP       T0912	// R_1-2 ROT R LMT RST TM
OR        D002220.2	// R_1st BD Z SERVO RESET
AND NOT   T0812	// R_1-2 ROT R RST TM
OUT       D002220.2	// R_1st BD Z SERVO RESET
TON       T0812 1	// R_1-2 ROT R RST TM
; L235
LOAD      F00099
DMOV      D004282 D002228	// R_1st ROT X Á¶±×Àú¼Ó
// Currnent Postition
; L237
LOADD=    D004240 D001226	// R_1st BD Z UP POS
AND       T0512	// R_1-2 ROT R READY
AND       M01622
OUT       M04120	// R_1-2 ROT R IDLE POS
; L238
LOADD=    D004242 D001226	// R_1st BD Z CENTER POS
AND       T0512	// R_1-2 ROT R READY
AND       M01622
OUT       M04121	// R_1-2 ROT R ROT POS
; L239
LOADD=    D004244 D001226	// R_1st BD Z BD POS
AND       T0512	// R_1-2 ROT R READY
AND       M01622
OUT       M04122	// R_1-2 ROT R BACK POS
; L240
LOAD      F00099
DADD      D004240 D004258 D004242	// R_1st BD Z UP POS / R_1st BD Z CENTER POS
; L241
END

PROGRAM 54_MT_13_14_15_16 (task: ½ºÄµ ÇÁ·Î±×·¥)

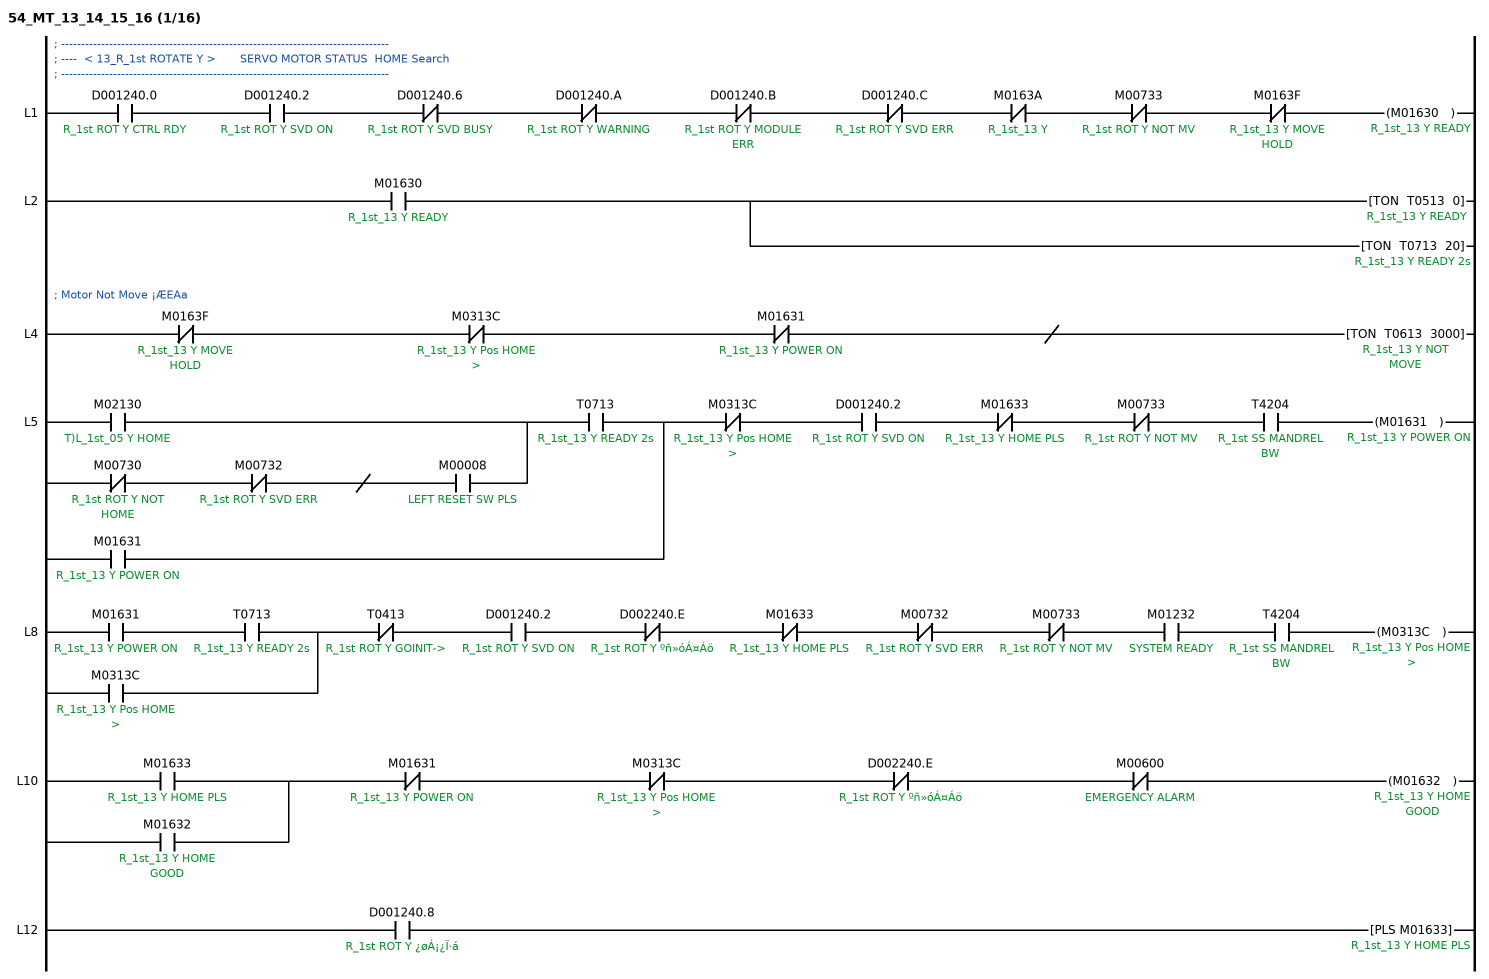
// ----------------------------------------------------------------------------------
// 
// ----  < 13_R_1st ROTATE Y >       SERVO MOTOR STATUS  HOME Search
// 
// ----------------------------------------------------------------------------------
; L1
LOAD      D001240.0	// R_1st ROT Y CTRL RDY
AND       D001240.2	// R_1st ROT Y SVD ON
AND NOT   D001240.6	// R_1st ROT Y SVD BUSY
AND NOT   D001240.A	// R_1st ROT Y WARNING
AND NOT   D001240.B	// R_1st ROT Y MODULE ERR
AND NOT   D001240.C	// R_1st ROT Y SVD ERR
AND NOT   M0163A	// R_1st_13 Y
AND NOT   M00733	// R_1st ROT Y NOT MV
AND NOT   M0163F	// R_1st_13 Y MOVE HOLD
OUT       M01630	// R_1st_13 Y READY
; L2
LOAD      M01630	// R_1st_13 Y READY
TON       T0513 0	// R_1st_13 Y READY
TON       T0713 20	// R_1st_13 Y READY 2s
; L4
LOAD NOT  M0163F	// R_1st_13 Y MOVE HOLD
AND NOT   M0313C	// R_1st_13 Y Pos HOME >
AND NOT   M01631	// R_1st_13 Y POWER ON
NOT
TON       T0613 3000	// R_1st_13 Y NOT MOVE
// output comment: Motor Not Move ¡ÆEAa
; L5
LOAD      M02130	// T)L_1st_05 Y HOME
LOAD NOT  M00730	// R_1st ROT Y NOT HOME
AND NOT   M00732	// R_1st ROT Y SVD ERR
NOT
AND       M00008	// LEFT RESET SW PLS
OR LOAD
AND       T0713	// R_1st_13 Y READY 2s
OR        M01631	// R_1st_13 Y POWER ON
AND NOT   M0313C	// R_1st_13 Y Pos HOME >
AND       D001240.2	// R_1st ROT Y SVD ON
AND NOT   M01633	// R_1st_13 Y HOME PLS
AND NOT   M00733	// R_1st ROT Y NOT MV
AND       T4204	// R_1st SS MANDREL BW
OUT       M01631	// R_1st_13 Y POWER ON
; L8
LOAD      M01631	// R_1st_13 Y POWER ON
AND       T0713	// R_1st_13 Y READY 2s
OR        M0313C	// R_1st_13 Y Pos HOME >
AND NOT   T0413	// R_1st ROT Y GOINIT->
AND       D001240.2	// R_1st ROT Y SVD ON
AND NOT   D002240.E	// R_1st ROT Y ºñ»óÁ¤Áö
AND NOT   M01633	// R_1st_13 Y HOME PLS
AND NOT   M00732	// R_1st ROT Y SVD ERR
AND NOT   M00733	// R_1st ROT Y NOT MV
AND       M01232	// SYSTEM READY
AND       T4204	// R_1st SS MANDREL BW
OUT       M0313C	// R_1st_13 Y Pos HOME >
; L10
LOAD      M01633	// R_1st_13 Y HOME PLS
OR        M01632	// R_1st_13 Y HOME GOOD
AND NOT   M01631	// R_1st_13 Y POWER ON
AND NOT   M0313C	// R_1st_13 Y Pos HOME >
AND NOT   D002240.E	// R_1st ROT Y ºñ»óÁ¤Áö
AND NOT   M00600	// EMERGENCY ALARM
OUT       M01632	// R_1st_13 Y HOME GOOD
; L12
LOAD      D001240.8	// R_1st ROT Y ¿øÁ¡¿Ï·á
OUTP      M01633	// R_1st_13 Y HOME PLS

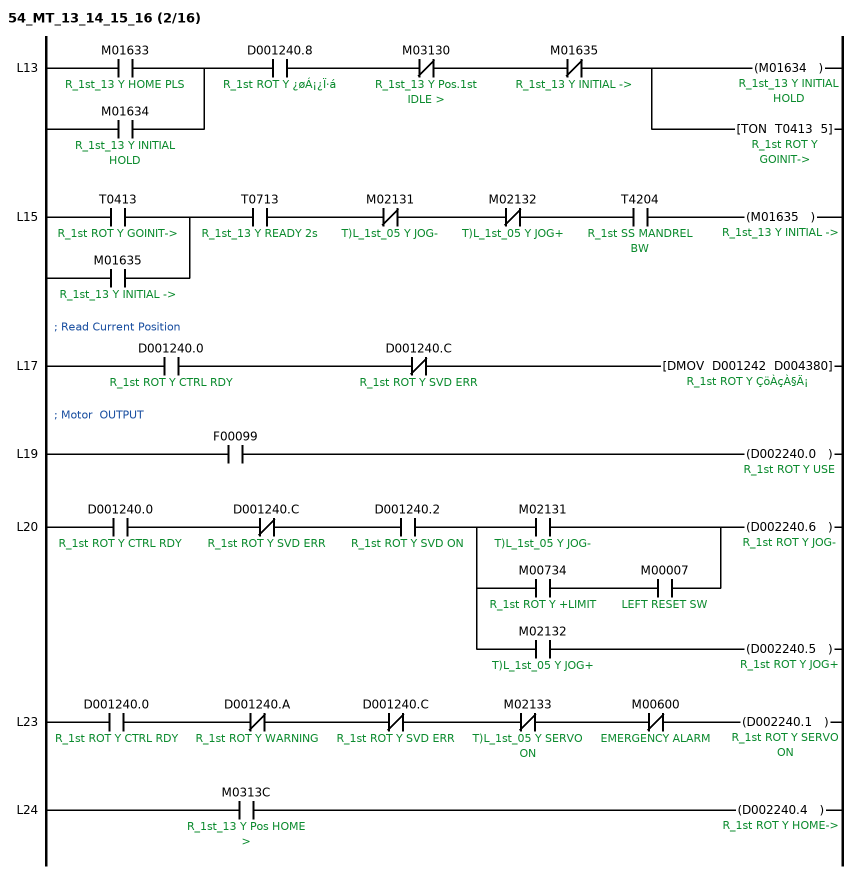
; L13
LOAD      M01633	// R_1st_13 Y HOME PLS
OR        M01634	// R_1st_13 Y INITIAL HOLD
AND       D001240.8	// R_1st ROT Y ¿øÁ¡¿Ï·á
AND NOT   M03130	// R_1st_13 Y Pos.1st IDLE >
AND NOT   M01635	// R_1st_13 Y INITIAL ->
OUT       M01634	// R_1st_13 Y INITIAL HOLD
TON       T0413 5	// R_1st ROT Y GOINIT->
; L15
LOAD      T0413	// R_1st ROT Y GOINIT->
OR        M01635	// R_1st_13 Y INITIAL ->
AND       T0713	// R_1st_13 Y READY 2s
AND NOT   M02131	// T)L_1st_05 Y JOG-
AND NOT   M02132	// T)L_1st_05 Y JOG+
AND       T4204	// R_1st SS MANDREL BW
OUT       M01635	// R_1st_13 Y INITIAL ->
; L17
LOAD      D001240.0	// R_1st ROT Y CTRL RDY
AND NOT   D001240.C	// R_1st ROT Y SVD ERR
DMOV      D001242 D004380	// R_1st ROT Y ÇöÀçÀ§Ä¡
// output comment: Read Current Position
//  Motor  OUTPUT
; L19
LOAD      F00099
OUT       D002240.0	// R_1st ROT Y USE
; L20
LOAD      D001240.0	// R_1st ROT Y CTRL RDY
AND NOT   D001240.C	// R_1st ROT Y SVD ERR
AND       D001240.2	// R_1st ROT Y SVD ON
MPUSH
LOAD      M02131	// T)L_1st_05 Y JOG-
LOAD      M00734	// R_1st ROT Y +LIMIT
AND       M00007	// LEFT RESET SW
OR LOAD
AND LOAD
OUT       D002240.6	// R_1st ROT Y JOG-
MPOP
AND       M02132	// T)L_1st_05 Y JOG+
OUT       D002240.5	// R_1st ROT Y JOG+
; L23
LOAD      D001240.0	// R_1st ROT Y CTRL RDY
AND NOT   D001240.A	// R_1st ROT Y WARNING
AND NOT   D001240.C	// R_1st ROT Y SVD ERR
AND NOT   M02133	// T)L_1st_05 Y SERVO ON
AND NOT   M00600	// EMERGENCY ALARM
OUT       D002240.1	// R_1st ROT Y SERVO ON
; L24
LOAD      M0313C	// R_1st_13 Y Pos HOME >
OUT       D002240.4	// R_1st ROT Y HOME->

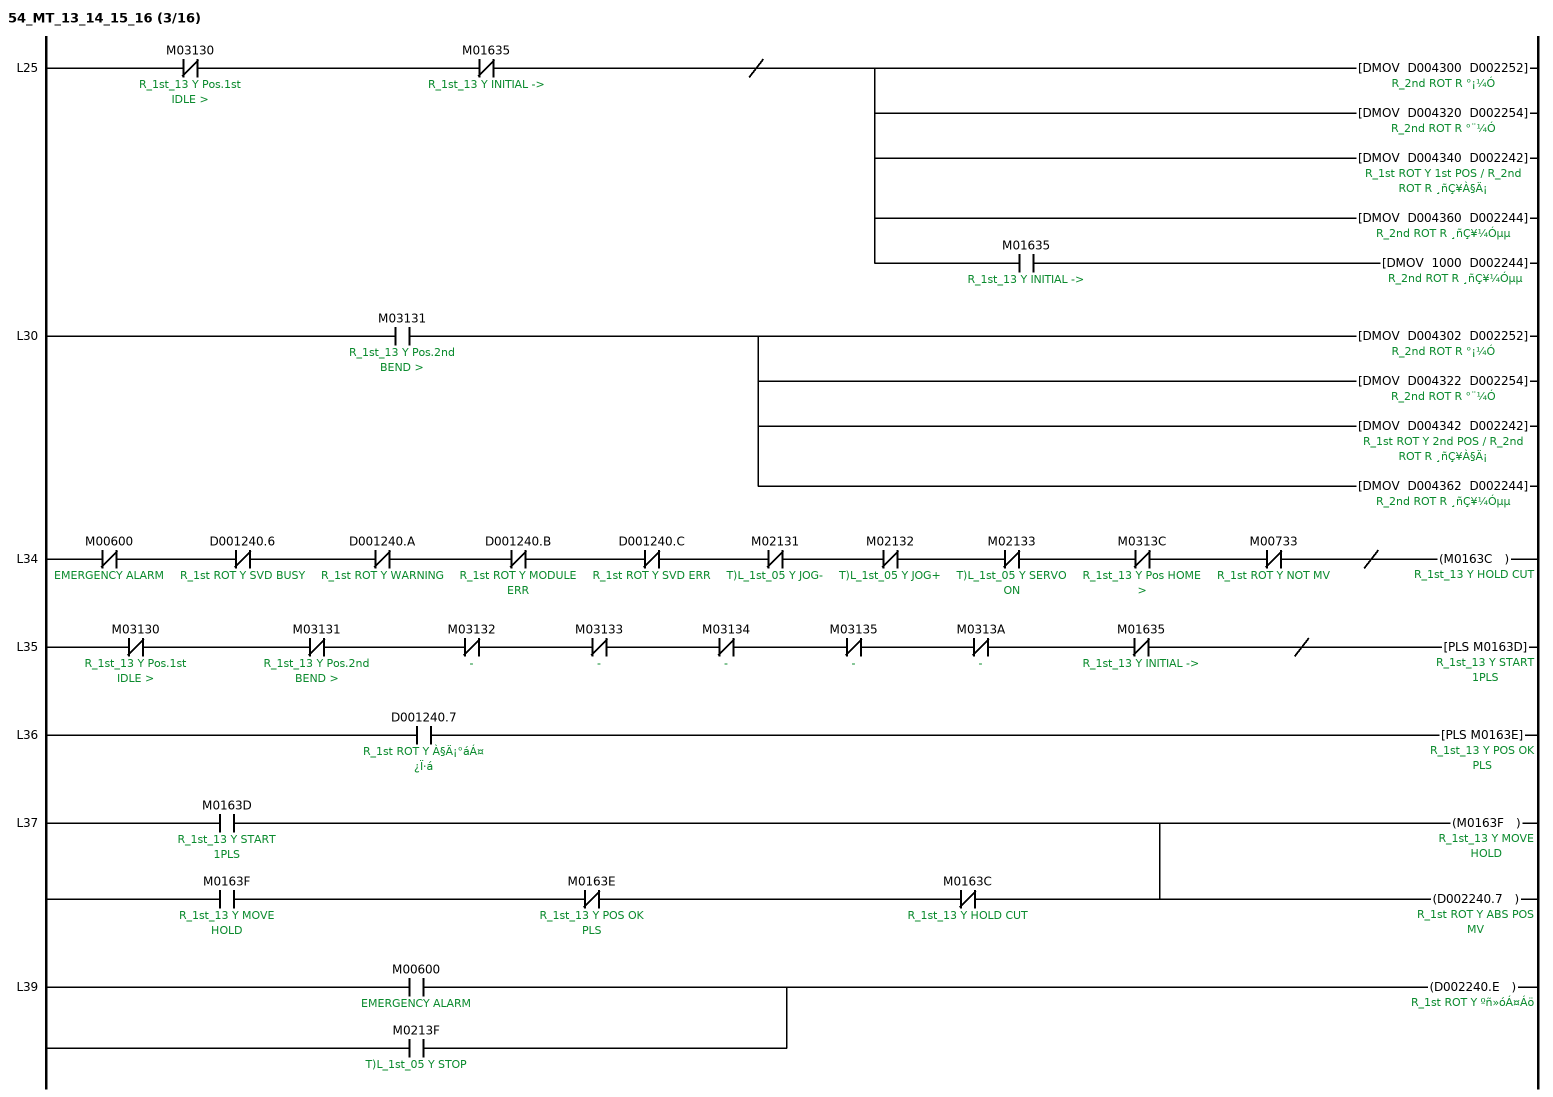
; L25
LOAD NOT  M03130	// R_1st_13 Y Pos.1st IDLE >
AND NOT   M01635	// R_1st_13 Y INITIAL ->
NOT
DMOV      D004300 D002252	// R_2nd ROT R °¡¼Ó
DMOV      D004320 D002254	// R_2nd ROT R °¨¼Ó
DMOV      D004340 D002242	// R_1st ROT Y 1st POS / R_2nd ROT R ¸ñÇ¥À§Ä¡
DMOV      D004360 D002244	// R_2nd ROT R ¸ñÇ¥¼Óµµ
AND       M01635	// R_1st_13 Y INITIAL ->
DMOV      1000 D002244	// R_2nd ROT R ¸ñÇ¥¼Óµµ
; L30
LOAD      M03131	// R_1st_13 Y Pos.2nd BEND >
DMOV      D004302 D002252	// R_2nd ROT R °¡¼Ó
DMOV      D004322 D002254	// R_2nd ROT R °¨¼Ó
DMOV      D004342 D002242	// R_1st ROT Y 2nd POS / R_2nd ROT R ¸ñÇ¥À§Ä¡
DMOV      D004362 D002244	// R_2nd ROT R ¸ñÇ¥¼Óµµ
; L34
LOAD NOT  M00600	// EMERGENCY ALARM
AND NOT   D001240.6	// R_1st ROT Y SVD BUSY
AND NOT   D001240.A	// R_1st ROT Y WARNING
AND NOT   D001240.B	// R_1st ROT Y MODULE ERR
AND NOT   D001240.C	// R_1st ROT Y SVD ERR
AND NOT   M02131	// T)L_1st_05 Y JOG-
AND NOT   M02132	// T)L_1st_05 Y JOG+
AND NOT   M02133	// T)L_1st_05 Y SERVO ON
AND NOT   M0313C	// R_1st_13 Y Pos HOME >
AND NOT   M00733	// R_1st ROT Y NOT MV
NOT
OUT       M0163C	// R_1st_13 Y HOLD CUT
; L35
LOAD NOT  M03130	// R_1st_13 Y Pos.1st IDLE >
AND NOT   M03131	// R_1st_13 Y Pos.2nd BEND >
AND NOT   M03132	// -
AND NOT   M03133	// -
AND NOT   M03134	// -
AND NOT   M03135	// -
AND NOT   M0313A	// -
AND NOT   M01635	// R_1st_13 Y INITIAL ->
NOT
OUTP      M0163D	// R_1st_13 Y START 1PLS
; L36
LOAD      D001240.7	// R_1st ROT Y À§Ä¡°áÁ¤ ¿Ï·á
OUTP      M0163E	// R_1st_13 Y POS OK PLS
; L37
LOAD      M0163D	// R_1st_13 Y START 1PLS
LOAD      M0163F	// R_1st_13 Y MOVE HOLD
AND NOT   M0163E	// R_1st_13 Y POS OK PLS
AND NOT   M0163C	// R_1st_13 Y HOLD CUT
OR LOAD
OUT       M0163F	// R_1st_13 Y MOVE HOLD
OUT       D002240.7	// R_1st ROT Y ABS POS MV
; L39
LOAD      M00600	// EMERGENCY ALARM
OR        M0213F	// T)L_1st_05 Y STOP
OUT       D002240.E	// R_1st ROT Y ºñ»óÁ¤Áö

